// TwinCAT 3 PLC project ST710
// ProgramVersion: 3.1.4024.0
// libraries:
//   Tc2_Standard, * (Beckhoff Automation GmbH)
//   Tc2_System, * (Beckhoff Automation GmbH)
//   Tc3_Module, * (Beckhoff Automation GmbH)
// project tree:
//   DUTs/ Cyl_Module_DUT.TcDUT
//   / GlobalTextList.TcGTLO, PlcTask.TcTTO, Visualization Manager.TcVMO (not stored)
//   GVLs/ Alarm_DB.TcGVL, Auto_Seq_DB.TcGVL, Home_Seq_DB.TcGVL, Inputs.TcGVL, Outputs.TcGVL, Stn710_DB.TcGVL
//   POUs/ Auto_Sequence.TcPOU, HomeSequence.TcPOU, MAIN.TcPOU, Alarms.TcPOU, Robot.TcPOU, Module_call.TcPOU, PowerOn.TcPOU, RollerDoor.TcPOU, Trunion.TcPOU, TurnTable.TcPOU
//   POUs/Library/ Seq_list.TcTLO, FB_CylinderModule.TcPOU, Feedback_FB.TcPOU, Alarm_list.TcTLO
//   VISUs/ Visualization.TcVIS
// real-time tasks:
//   TASK PlcTask: cycle T#10ms, priority 20, ADS port 350

CONFIGURATION ST710
    RESOURCE PLC ON TwinCAT3
        TASK PlcTask(INTERVAL := T#10ms, PRIORITY := 20);
        PROGRAM MAIN WITH PlcTask : MAIN;
    END_RESOURCE
END_CONFIGURATION

// ---- DUTs/Cyl_Module_DUT.TcDUT
TYPE Cyl_Module_DUT :
STRUCT
	ResetFaults:BOOL;//Reset Fault CMD
    WorkCmd:BOOL ;//Cyl Work Postion CMD
    HomeCmd:BOOL ;//Cyl Home Postion CMD
    WorkSen:BOOL ;// Cyl Work Postion Input
    HomeSen:BOOL ;// Cyl Home Postion Input
    WorkCleartoMove:BOOL ;// Condition Healthy then 1
    HomeCleartoMove:BOOL ;// Condition Healthy then 1
    TimeoutValue:TIME ;// Time Required E.gT#500MS,T#2S
	ENO   : BOOL; //  Block Enable
	WorkSol    : BOOL; // Cyl Work Position Sol Output
    HomeSol: BOOL; //Cyl Home Position Sol Output
    WorkOver: BOOL; // Cyl AT Work Position
    HomeOver: BOOL; //Cyl AT Home Position
    ErrHomeInterlock: BOOL; //homeCleartoMove is low AND home command is active.
    ErrHomeTout: BOOL; //cylinder did NOT reachhome position within definedTIME
    ErrWorkInterlock: BOOL; //WorkCleartoMove is low AND work command is active.
    ErrWorkTout: BOOL; //cylinder did NOT reachwork position within definedtime
END_STRUCT
END_TYPE

// ---- GVLs/Alarm_DB.TcGVL
{attribute 'qualified_only'}
VAR_GLOBAL
	EMR_Stop_pressed : BOOL;
END_VAR

// ---- GVLs/Auto_Seq_DB.TcGVL
{attribute 'qualified_only'}
VAR_GLOBAL
	MHomeCycleStart		:BOOL;
	MWELD_RobotStart	:BOOL;
	M_MH_RobotStart		:BOOL;
	MCycleRun			:BOOL;
	MRollerDoor_CLOSE	:BOOL;
	MRollerDoor_Open	:BOOL;
	MTrunion_Move_0		:BOOL;
	MTrunion_Move_20	:BOOL;
	MTrunion_Move_45	:BOOL;
	MTrunion_Move_80	:BOOL;
	MClampClsGroup1		:BOOL;
	MClampClsGroup2		:BOOL;
	MTurntable_0		:BOOL;
	MTurntable_180		:BOOL;
	MClampOpenGrp1		:BOOL;
	MClampOpenGrp2		:BOOL;
	MStep				:INT;
	Part_Sensor1		:BOOL;
	Part_Sensor2		:BOOL;
	Part_Sensor3		:BOOL;
	Part_Sensor4		:BOOL;
END_VAR

// ---- GVLs/Home_Seq_DB.TcGVL
{attribute 'qualified_only'}
VAR_GLOBAL
	M_Group1ClampOpen :BOOL;
	M_Group2ClampOpen :BOOL;
	M_TT_0 : BOOL;
	M_Trunion_0 : BOOL;
	M_Door_Cls : BOOL;
	M_HomeDone : Bool;
END_VAR

// ---- GVLs/Inputs.TcGVL
{attribute 'qualified_only'}
VAR_GLOBAL
	Control_Pressure_Sw_In1_BPB1	: BOOL ;
	Control_Pressure_Sw_In2_BPB1	: BOOL ;
	Valve_Pos_BGB1					: BOOL ;
	CC6_Clamp_1_Sensor_HP			: BOOL ;
	CC6_Clamp_1_Sensor_WP			: BOOL ;
	CC4_Clamp_3_Sensor_HP			: BOOL ;
	CC4_Clamp_3_Sensor_WP			: BOOL ;
	CC4_Clamp_2_Sensor_HP			: BOOL ;
	CC4_Clamp_2_Sensor_WP			: BOOL ;
	CC4_Clamp_1_Sensor_HP			: BOOL ;
	CC4_Clamp_1_Sensor_WP			: BOOL ;
	CC2_Clamp_3_Sensor_HP			: BOOL ;
	CC2_Clamp_3_Sensor_WP			: BOOL ;
	CC3_Clamp_3_Sensor_HP			: BOOL ;
	CC3_Clamp_3_Sensor_WP			: BOOL ;
	CC3_Clamp_2_Sensor_HP			: BOOL ;
	CC3_Clamp_2_Sensor_WP			: BOOL ;
	CC3_Clamp_1_Sensor_HP			: BOOL ;
	CC3_Clamp_1_Sensor_WP			: BOOL ;
	CC1_Clamp_3_Sensor_HP			: BOOL ;
	CC1_Clamp_3_Sensor_WP			: BOOL ;
	CC1_Clamp_2_Sensor_HP			: BOOL ;
	CC1_Clamp_2_Sensor_WP			: BOOL ;
	CC1_Clamp_1_Sensor_HP			: BOOL ;
	CC1_Clamp_1_Sensor_WP			: BOOL ;
	CC2_Clamp_2_Sensor_HP			: BOOL ;
	CC2_Clamp_2_Sensor_WP			: BOOL ;
	CC2_Clamp_1_Sensor_HP			: BOOL ;
	CC2_Clamp_1_Sensor_WP			: BOOL ;
	CC5_Clamp_1_Sensor_HP			: BOOL ;
	CC5_Clamp_1_Sensor_WP			: BOOL ;
	PART_CONTROL_B13				: BOOL ;
	PART_CONTROL_B27				: BOOL ;
	PART_CONTROL_B14				: BOOL ;
	PART_CONTROL_B28				: BOOL ;
	PART_CONTROL_B12				: BOOL ;
	PART_CONTROL_B26				: BOOL ;
	PART_CONTROL_B11				: BOOL ;
	PART_CONTROL_B25				: BOOL ;
	PART_CONTROL_B10				: BOOL ;
	PART_CONTROL_B24				: BOOL ;
	PART_CONTROL_B7					: BOOL ;
	PART_CONTROL_B21				: BOOL ;
	PART_CONTROL_B6					: BOOL ;
	PART_CONTROL_B20				: BOOL ;
	PART_CONTROL_B5					: BOOL ;
	PART_CONTROL_B19				: BOOL ;
	PART_CONTROL_B4			 		: BOOL ;
	PART_CONTROL_B18				: BOOL ;
	PART_CONTROL_B3					: BOOL ;
	PART_CONTROL_B17				: BOOL ;
	PART_CONTROL_B2					: BOOL ;
	PART_CONTROL_B9					: BOOL ;
	PART_CONTROL_B23				: BOOL ;
	PART_CONTROL_B8					: BOOL ;
	PART_CONTROL_B22				: BOOL ;
	iEMR_Stop_PB					: BOOL ;
	iControl_On						: BOOL ;
	iControl_Off					: BOOL ;
	iAuto_Manual					: BOOL ;
	iResetFault 					: BOOL ;
	iCycle_start					:BOOL;
	iPalm_Button					:BOOL;
	
END_VAR

// ---- GVLs/Outputs.TcGVL
{attribute 'qualified_only'}
VAR_GLOBAL
	CC1_CLAMPING_UNIT1_3_WP			: BOOL ;
	CC1_CLAMPING_UNIT1_3_HP			: BOOL ;
	CC2_CLAMPING_UNIT2_3_WP			: BOOL ;
	CC2_CLAMPING_UNIT2_3_HP			: BOOL ;
	CC3_CLAMPING_UNIT3_3_WP			: BOOL ;
	CC3_CLAMPING_UNIT3_3_HP			: BOOL ;
	CC4_CLAMPING_UNIT4_3_WP			: BOOL ;
	CC4_CLAMPING_UNIT4_3_HP			: BOOL ;
	CC5_CLAMPING_UNIT5_1_WP			: BOOL ;
	CC5_CLAMPING_UNIT5_1_HP			: BOOL ;
	CC6_CLAMPING_UNIT6_1_WP			: BOOL ;
	CC6_CLAMPING_UNIT6_1_HP			: BOOL ;
	qPower_On						: BOOL ;
	qStnAuto						: BOOL ;
	qStnMan							: BOOL ;
END_VAR

// ---- GVLs/Stn710_DB.TcGVL
{attribute 'qualified_only'}
VAR_GLOBAL
	M_TT_MotorRun  : BOOL;
	M_TT_MotorDir  : BOOL;
	M_TT_CW		   : BOOL;
	M_TT_CCW		: BOOL;
	M_TT_FwdSens	: BOOL;
	M_TT_RevSens	: BOOL;
	M_TR_Motor0  	: BOOL;
	M_TR_Motor20  	: BOOL;
	M_TR_Motor45  	: BOOL;
	M_TR_Motor80  	: BOOL;
	M_TR_0_FB		: BOOL;
	M_TR_20_FB		: BOOL;
	M_TR_45_FB		: BOOL;
	M_TR_80_FB		: BOOL;
	M_TR_0_CMD		: BOOL;
	M_TR_20_CMD		: BOOL;
	M_TR_45_CMD		: BOOL;
	M_TR_80_CMD		: BOOL;
	MQ_DR_UP	  	: BOOL;
	MQ_DR_DOWN  	: BOOL;
	M_DR_UP		   	: BOOL;
	M_DR_DOWN		: BOOL;
	M_DR_UPSens		: BOOL;
	M_DR_DNSens		: BOOL;
	MH_RobotHome	: BOOL;
	MH_RobotBusy	: BOOL;
	MH_RobotDone	: BOOL;
	WELD_RobotHome	: BOOL;
	WELD_RobotBusy	: BOOL;
	WELD_RobotDone	: BOOL;
	Alarm_count : INT;
	CC1_CLAMP : Cyl_Module_DUT;
	CC2_CLAMP : Cyl_Module_DUT;
	CC3_CLAMP : Cyl_Module_DUT;
	CC4_CLAMP : Cyl_Module_DUT;
	CC5_CLAMP : Cyl_Module_DUT;
	CC6_CLAMP : Cyl_Module_DUT;	
END_VAR

// ---- POUs/MAIN.TcPOU
PROGRAM MAIN
VAR
	Modules: Module_call;
	tAlwaysOn: BOOL; //Temporary BIT FOR Always On
    tAlwaysOff: BOOL; //Temporary BIT FOR Always Off
END_VAR

VAR CONSTANT
END_VAR

// Always ON Logic
tAlwaysOn := TRUE;

// Module call
Modules();

END_PROGRAM

// ---- POUs/Module_call.TcPOU
FUNCTION_BLOCK Module_call
VAR_INPUT
END_VAR
VAR_OUTPUT
END_VAR
VAR
	CC1_UNIT1_3_Cyl: FB_CylinderModule;	
	CC2_UNIT2_3_Cyl: FB_CylinderModule;
	CC3_UNIT3_3_Cyl: FB_CylinderModule;
	CC4_UNIT4_3_Cyl: FB_CylinderModule;
	CC5_UNIT5_1_Cyl: FB_CylinderModule;
	CC6_UNIT6_1_Cyl: FB_CylinderModule;
	CC1_Feedback_FB: Feedback_FB;
	CC2_Feedback_FB: Feedback_FB;
	CC3_Feedback_FB: Feedback_FB;
	CC4_Feedback_FB: Feedback_FB;
	CC5_Feedback_FB: Feedback_FB;
	CC6_Feedback_FB: Feedback_FB;
	CC1_Feedback_1: BOOL;
	CC1_Feedback_2: BOOL;
	CC2_Feedback_1: BOOL;
	CC2_Feedback_2: BOOL;
	CC3_Feedback_1: BOOL;
	CC3_Feedback_2: BOOL;
	CC4_Feedback_1: BOOL;
	CC4_Feedback_2: BOOL;
	PowerOn: PowerOn;
	TurnTable_0: TurnTable;
	TT_Feedback_FB: Feedback_FB;
	Trunion_0: Trunion;
	Tr_Feedback_FB: Feedback_FB;
	RollerDoor_0: RollerDoor;
	Door_Feedback_FB: Feedback_FB;
	MH_Robot: Robot;
	Weld_Robot: Robot;
	Auto_Sequence_0: Auto_Sequence;
	TR_Feedback_FB1: Feedback_FB;
	HomeSequence_0: HomeSequence;
	Alarms_0: Alarms;
END_VAR
VAR // added by the converter: edge detectors and wires of the graphical bodies
    _w1, _w2, _w3, _w4, _w5, _w6, _w7, _w8 : BOOL;
END_VAR

// note: this text did not pass the execution check against the stored diagram
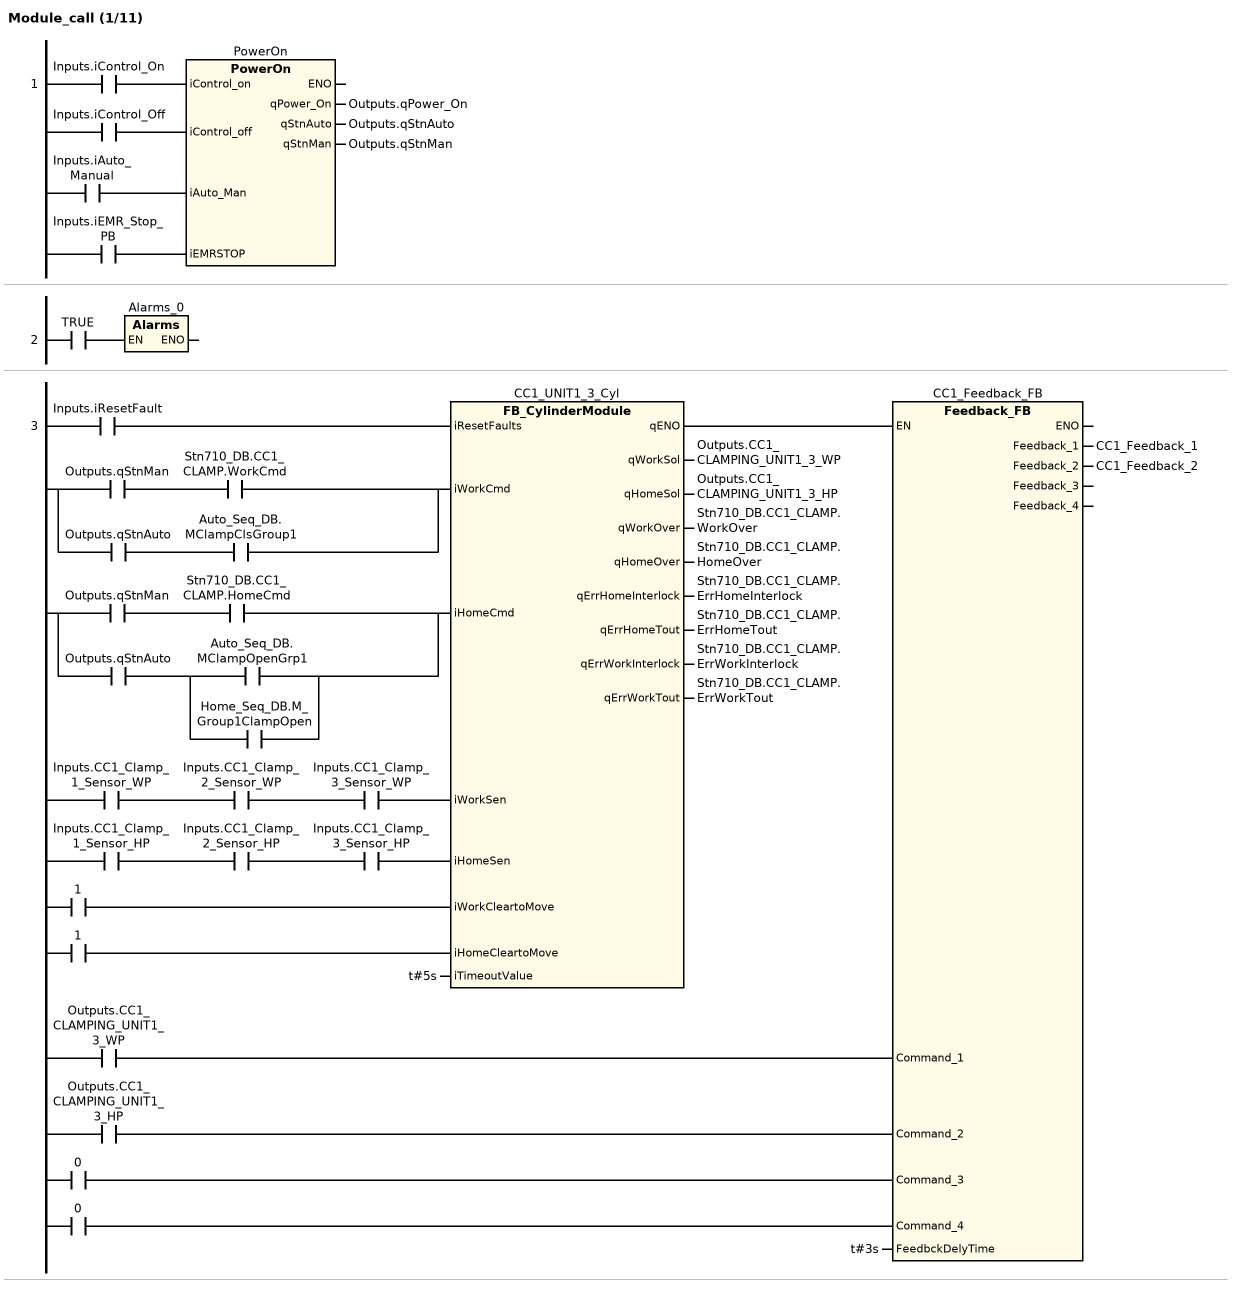
// NETWORK 1
PowerOn(
    iControl_on := Inputs.iControl_On,
    iControl_off := Inputs.iControl_Off,
    iAuto_Man := Inputs.iAuto_Manual,
    iEMRSTOP := Inputs.iEMR_Stop_PB,
    qPower_On => Outputs.qPower_On,
    qStnAuto => Outputs.qStnAuto,
    qStnMan => Outputs.qStnMan);

// NETWORK 2
Alarms_0(EN := TRUE); // Alarms

// NETWORK 3
CC1_UNIT1_3_Cyl(
    iResetFaults := Inputs.iResetFault,
    iWorkCmd := Outputs.qStnMan AND Stn710_DB.CC1_CLAMP.WorkCmd OR Outputs.qStnAuto AND Auto_Seq_DB.MClampClsGroup1,
    iHomeCmd := Outputs.qStnMan AND Stn710_DB.CC1_CLAMP.HomeCmd OR Outputs.qStnAuto AND (Auto_Seq_DB.MClampOpenGrp1 OR Home_Seq_DB.M_Group1ClampOpen),
    iWorkSen := Inputs.CC1_Clamp_1_Sensor_WP AND Inputs.CC1_Clamp_2_Sensor_WP AND Inputs.CC1_Clamp_3_Sensor_WP,
    iHomeSen := Inputs.CC1_Clamp_1_Sensor_HP AND Inputs.CC1_Clamp_2_Sensor_HP AND Inputs.CC1_Clamp_3_Sensor_HP,
    iWorkCleartoMove := 1,
    iHomeCleartoMove := 1,
    iTimeoutValue := t#5s,
    qWorkSol => Outputs.CC1_CLAMPING_UNIT1_3_WP,
    qHomeSol => Outputs.CC1_CLAMPING_UNIT1_3_HP,
    qWorkOver => Stn710_DB.CC1_CLAMP.WorkOver,
    qHomeOver => Stn710_DB.CC1_CLAMP.HomeOver,
    qErrHomeInterlock => Stn710_DB.CC1_CLAMP.ErrHomeInterlock,
    qErrHomeTout => Stn710_DB.CC1_CLAMP.ErrHomeTout,
    qErrWorkInterlock => Stn710_DB.CC1_CLAMP.ErrWorkInterlock,
    qErrWorkTout => Stn710_DB.CC1_CLAMP.ErrWorkTout); // FB_CylinderModule
CC1_Feedback_FB(
    EN := CC1_UNIT1_3_Cyl.qENO,
    Command_1 := Outputs.CC1_CLAMPING_UNIT1_3_WP,
    Command_2 := Outputs.CC1_CLAMPING_UNIT1_3_HP,
    Command_3 := 0,
    Command_4 := 0,
    FeedbckDelyTime := t#3s,
    Feedback_1 => CC1_Feedback_1,
    Feedback_2 => CC1_Feedback_2); // Feedback_FB

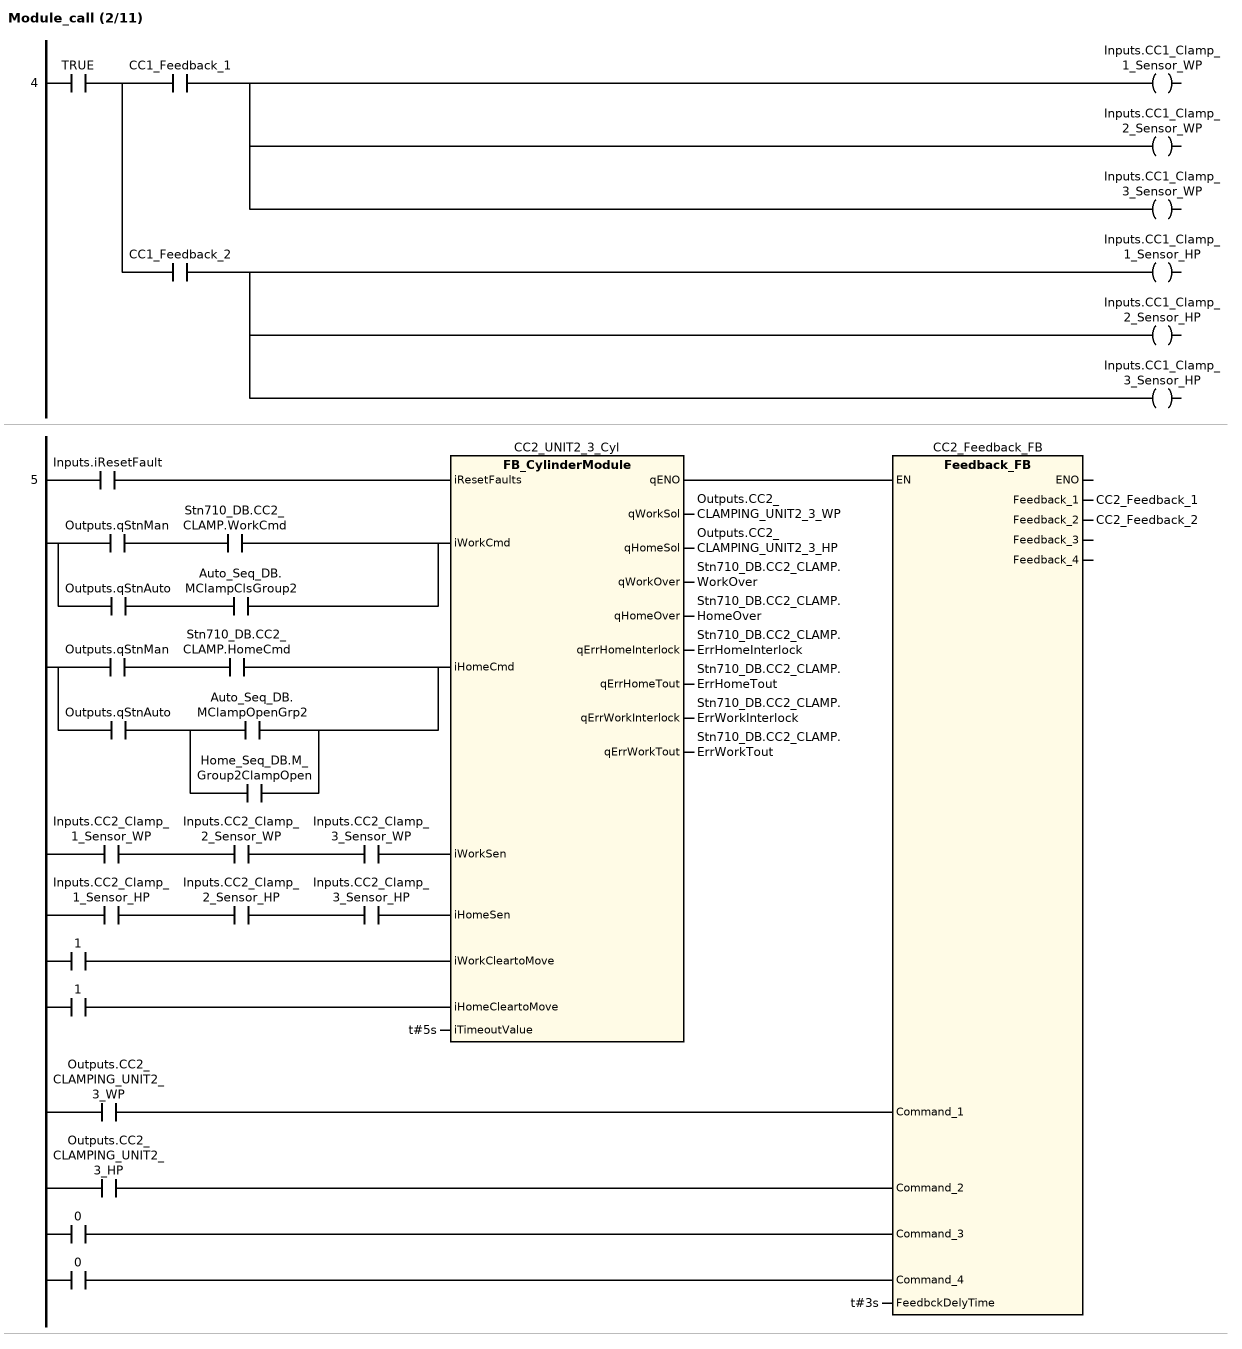
// NETWORK 4
_w1 := TRUE AND CC1_Feedback_1;
Inputs.CC1_Clamp_1_Sensor_WP := _w1;
Inputs.CC1_Clamp_2_Sensor_WP := _w1;
Inputs.CC1_Clamp_3_Sensor_WP := _w1;
_w2 := TRUE AND CC1_Feedback_2;
Inputs.CC1_Clamp_1_Sensor_HP := _w2;
Inputs.CC1_Clamp_2_Sensor_HP := _w2;
Inputs.CC1_Clamp_3_Sensor_HP := _w2;

// NETWORK 5
CC2_UNIT2_3_Cyl(
    iResetFaults := Inputs.iResetFault,
    iWorkCmd := Outputs.qStnMan AND Stn710_DB.CC2_CLAMP.WorkCmd OR Outputs.qStnAuto AND Auto_Seq_DB.MClampClsGroup2,
    iHomeCmd := Outputs.qStnMan AND Stn710_DB.CC2_CLAMP.HomeCmd OR Outputs.qStnAuto AND (Auto_Seq_DB.MClampOpenGrp2 OR Home_Seq_DB.M_Group2ClampOpen),
    iWorkSen := Inputs.CC2_Clamp_1_Sensor_WP AND Inputs.CC2_Clamp_2_Sensor_WP AND Inputs.CC2_Clamp_3_Sensor_WP,
    iHomeSen := Inputs.CC2_Clamp_1_Sensor_HP AND Inputs.CC2_Clamp_2_Sensor_HP AND Inputs.CC2_Clamp_3_Sensor_HP,
    iWorkCleartoMove := 1,
    iHomeCleartoMove := 1,
    iTimeoutValue := t#5s,
    qWorkSol => Outputs.CC2_CLAMPING_UNIT2_3_WP,
    qHomeSol => Outputs.CC2_CLAMPING_UNIT2_3_HP,
    qWorkOver => Stn710_DB.CC2_CLAMP.WorkOver,
    qHomeOver => Stn710_DB.CC2_CLAMP.HomeOver,
    qErrHomeInterlock => Stn710_DB.CC2_CLAMP.ErrHomeInterlock,
    qErrHomeTout => Stn710_DB.CC2_CLAMP.ErrHomeTout,
    qErrWorkInterlock => Stn710_DB.CC2_CLAMP.ErrWorkInterlock,
    qErrWorkTout => Stn710_DB.CC2_CLAMP.ErrWorkTout); // FB_CylinderModule
CC2_Feedback_FB(
    EN := CC2_UNIT2_3_Cyl.qENO,
    Command_1 := Outputs.CC2_CLAMPING_UNIT2_3_WP,
    Command_2 := Outputs.CC2_CLAMPING_UNIT2_3_HP,
    Command_3 := 0,
    Command_4 := 0,
    FeedbckDelyTime := t#3s,
    Feedback_1 => CC2_Feedback_1,
    Feedback_2 => CC2_Feedback_2); // Feedback_FB

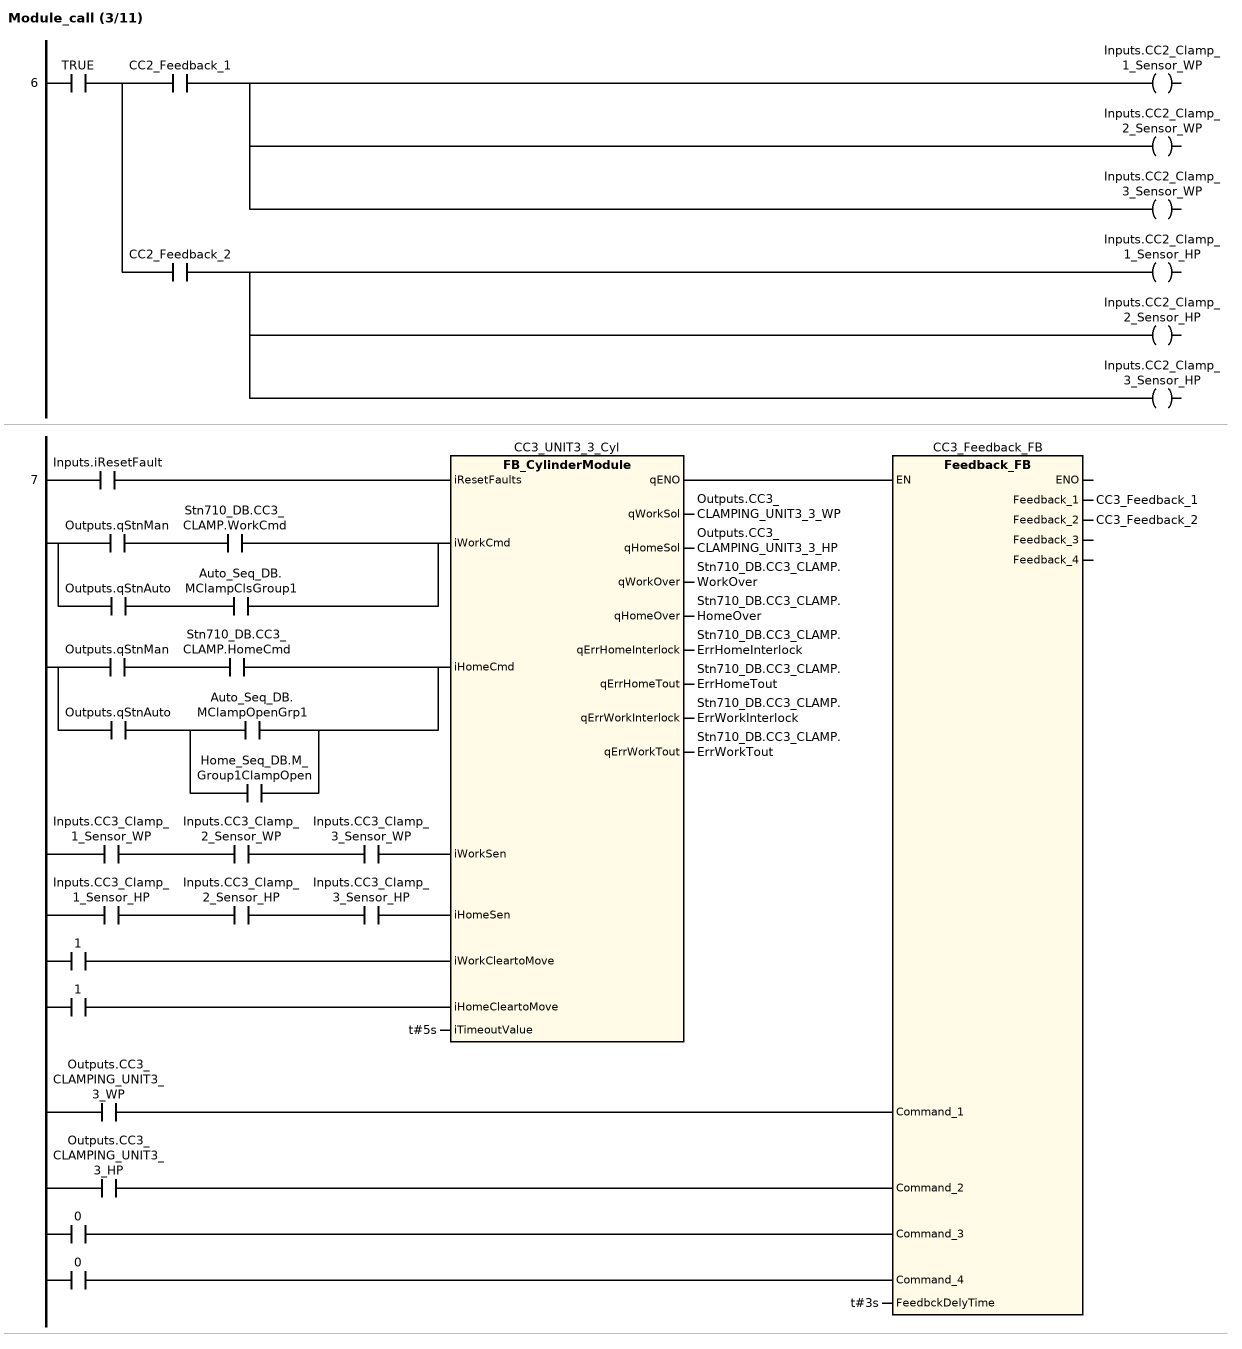
// NETWORK 6
_w3 := TRUE AND CC2_Feedback_1;
Inputs.CC2_Clamp_1_Sensor_WP := _w3;
Inputs.CC2_Clamp_2_Sensor_WP := _w3;
Inputs.CC2_Clamp_3_Sensor_WP := _w3;
_w4 := TRUE AND CC2_Feedback_2;
Inputs.CC2_Clamp_1_Sensor_HP := _w4;
Inputs.CC2_Clamp_2_Sensor_HP := _w4;
Inputs.CC2_Clamp_3_Sensor_HP := _w4;

// NETWORK 7
CC3_UNIT3_3_Cyl(
    iResetFaults := Inputs.iResetFault,
    iWorkCmd := Outputs.qStnMan AND Stn710_DB.CC3_CLAMP.WorkCmd OR Outputs.qStnAuto AND Auto_Seq_DB.MClampClsGroup1,
    iHomeCmd := Outputs.qStnMan AND Stn710_DB.CC3_CLAMP.HomeCmd OR Outputs.qStnAuto AND (Auto_Seq_DB.MClampOpenGrp1 OR Home_Seq_DB.M_Group1ClampOpen),
    iWorkSen := Inputs.CC3_Clamp_1_Sensor_WP AND Inputs.CC3_Clamp_2_Sensor_WP AND Inputs.CC3_Clamp_3_Sensor_WP,
    iHomeSen := Inputs.CC3_Clamp_1_Sensor_HP AND Inputs.CC3_Clamp_2_Sensor_HP AND Inputs.CC3_Clamp_3_Sensor_HP,
    iWorkCleartoMove := 1,
    iHomeCleartoMove := 1,
    iTimeoutValue := t#5s,
    qWorkSol => Outputs.CC3_CLAMPING_UNIT3_3_WP,
    qHomeSol => Outputs.CC3_CLAMPING_UNIT3_3_HP,
    qWorkOver => Stn710_DB.CC3_CLAMP.WorkOver,
    qHomeOver => Stn710_DB.CC3_CLAMP.HomeOver,
    qErrHomeInterlock => Stn710_DB.CC3_CLAMP.ErrHomeInterlock,
    qErrHomeTout => Stn710_DB.CC3_CLAMP.ErrHomeTout,
    qErrWorkInterlock => Stn710_DB.CC3_CLAMP.ErrWorkInterlock,
    qErrWorkTout => Stn710_DB.CC3_CLAMP.ErrWorkTout); // FB_CylinderModule
CC3_Feedback_FB(
    EN := CC3_UNIT3_3_Cyl.qENO,
    Command_1 := Outputs.CC3_CLAMPING_UNIT3_3_WP,
    Command_2 := Outputs.CC3_CLAMPING_UNIT3_3_HP,
    Command_3 := 0,
    Command_4 := 0,
    FeedbckDelyTime := t#3s,
    Feedback_1 => CC3_Feedback_1,
    Feedback_2 => CC3_Feedback_2); // Feedback_FB

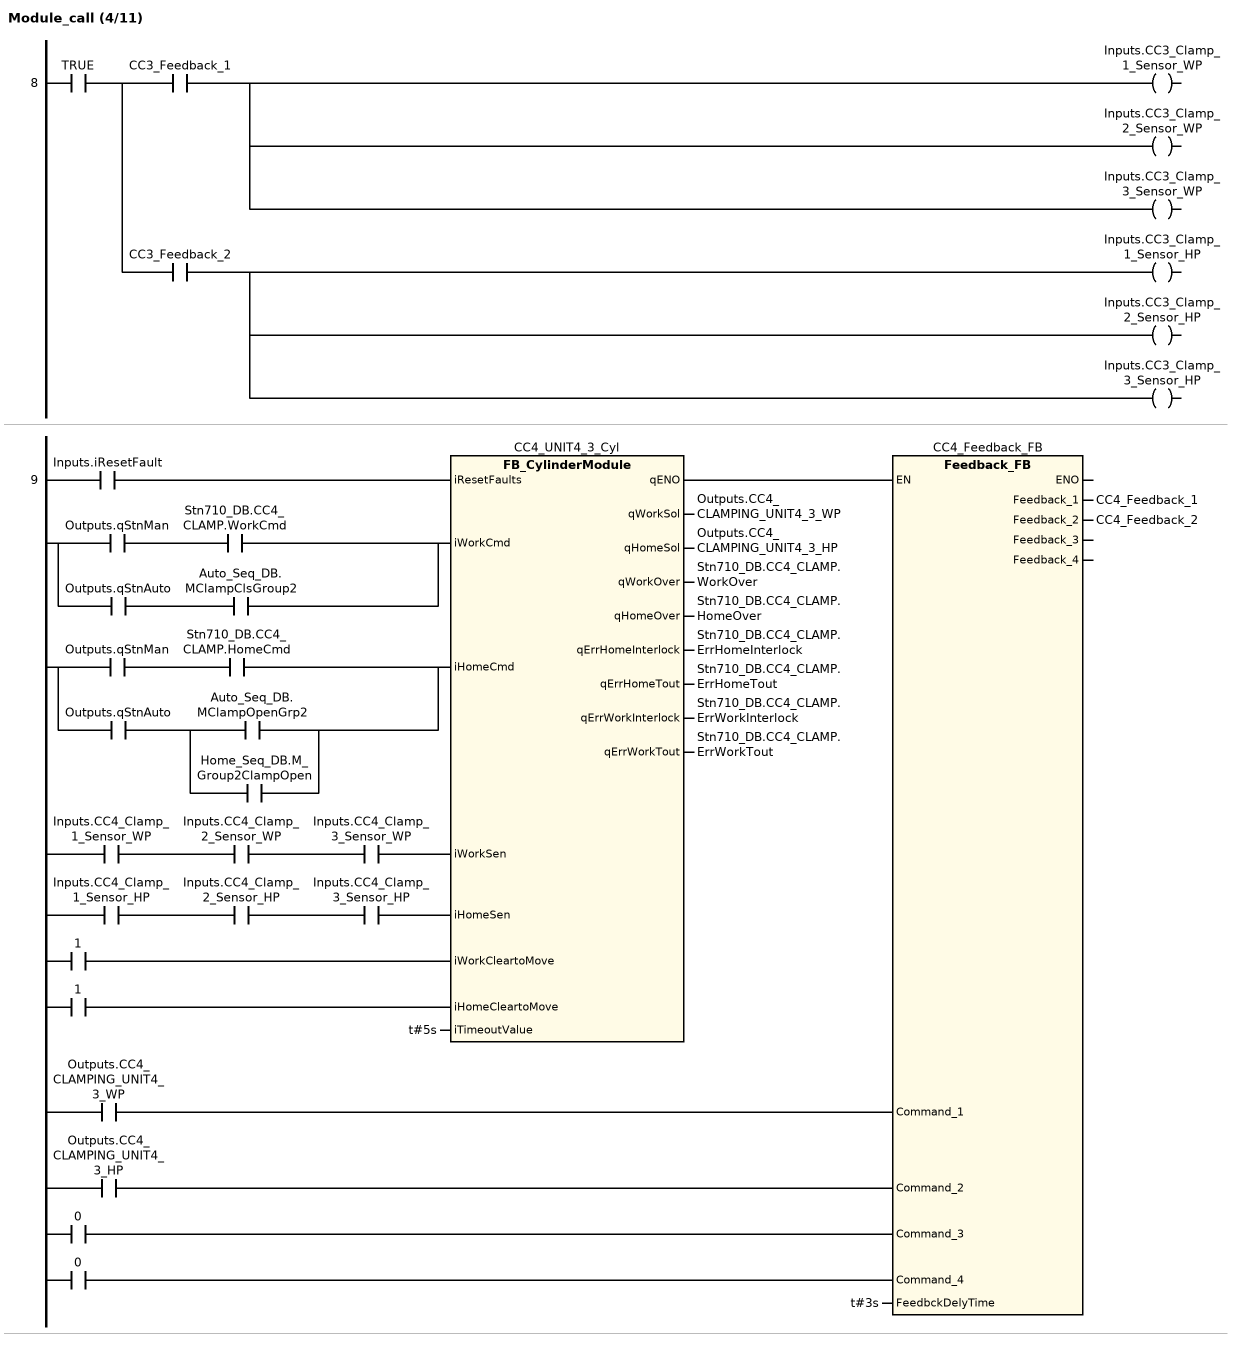
// NETWORK 8
_w5 := TRUE AND CC3_Feedback_1;
Inputs.CC3_Clamp_1_Sensor_WP := _w5;
Inputs.CC3_Clamp_2_Sensor_WP := _w5;
Inputs.CC3_Clamp_3_Sensor_WP := _w5;
_w6 := TRUE AND CC3_Feedback_2;
Inputs.CC3_Clamp_1_Sensor_HP := _w6;
Inputs.CC3_Clamp_2_Sensor_HP := _w6;
Inputs.CC3_Clamp_3_Sensor_HP := _w6;

// NETWORK 9
CC4_UNIT4_3_Cyl(
    iResetFaults := Inputs.iResetFault,
    iWorkCmd := Outputs.qStnMan AND Stn710_DB.CC4_CLAMP.WorkCmd OR Outputs.qStnAuto AND Auto_Seq_DB.MClampClsGroup2,
    iHomeCmd := Outputs.qStnMan AND Stn710_DB.CC4_CLAMP.HomeCmd OR Outputs.qStnAuto AND (Auto_Seq_DB.MClampOpenGrp2 OR Home_Seq_DB.M_Group2ClampOpen),
    iWorkSen := Inputs.CC4_Clamp_1_Sensor_WP AND Inputs.CC4_Clamp_2_Sensor_WP AND Inputs.CC4_Clamp_3_Sensor_WP,
    iHomeSen := Inputs.CC4_Clamp_1_Sensor_HP AND Inputs.CC4_Clamp_2_Sensor_HP AND Inputs.CC4_Clamp_3_Sensor_HP,
    iWorkCleartoMove := 1,
    iHomeCleartoMove := 1,
    iTimeoutValue := t#5s,
    qWorkSol => Outputs.CC4_CLAMPING_UNIT4_3_WP,
    qHomeSol => Outputs.CC4_CLAMPING_UNIT4_3_HP,
    qWorkOver => Stn710_DB.CC4_CLAMP.WorkOver,
    qHomeOver => Stn710_DB.CC4_CLAMP.HomeOver,
    qErrHomeInterlock => Stn710_DB.CC4_CLAMP.ErrHomeInterlock,
    qErrHomeTout => Stn710_DB.CC4_CLAMP.ErrHomeTout,
    qErrWorkInterlock => Stn710_DB.CC4_CLAMP.ErrWorkInterlock,
    qErrWorkTout => Stn710_DB.CC4_CLAMP.ErrWorkTout); // FB_CylinderModule
CC4_Feedback_FB(
    EN := CC4_UNIT4_3_Cyl.qENO,
    Command_1 := Outputs.CC4_CLAMPING_UNIT4_3_WP,
    Command_2 := Outputs.CC4_CLAMPING_UNIT4_3_HP,
    Command_3 := 0,
    Command_4 := 0,
    FeedbckDelyTime := t#3s,
    Feedback_1 => CC4_Feedback_1,
    Feedback_2 => CC4_Feedback_2); // Feedback_FB

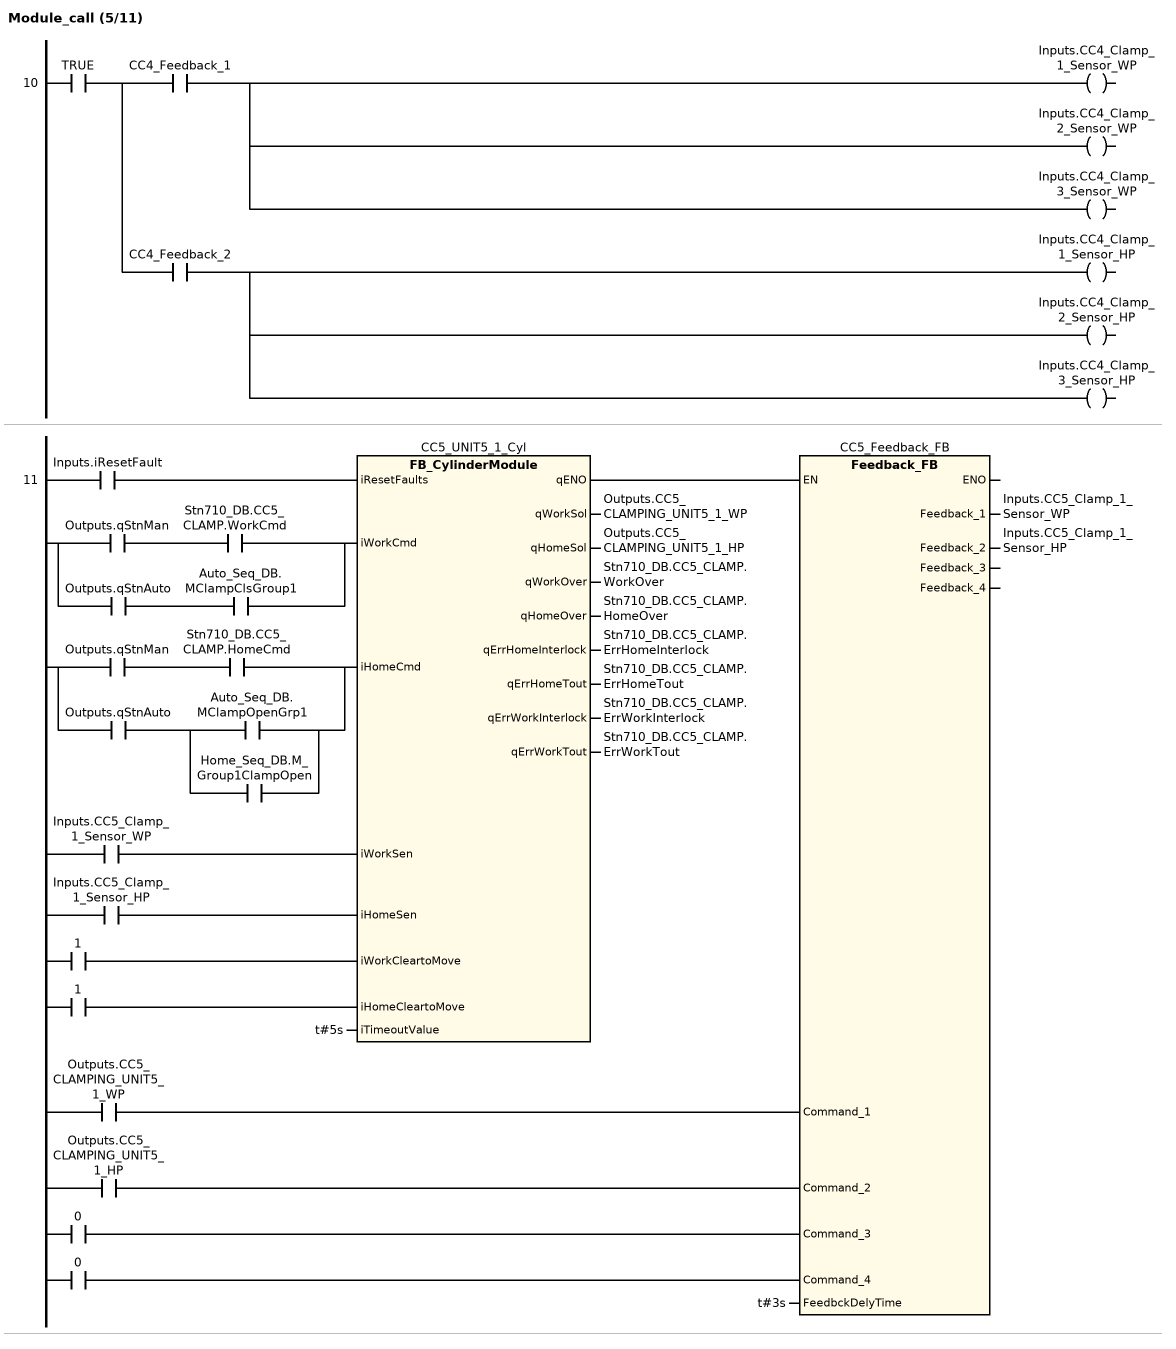
// NETWORK 10
_w7 := TRUE AND CC4_Feedback_1;
Inputs.CC4_Clamp_1_Sensor_WP := _w7;
Inputs.CC4_Clamp_2_Sensor_WP := _w7;
Inputs.CC4_Clamp_3_Sensor_WP := _w7;
_w8 := TRUE AND CC4_Feedback_2;
Inputs.CC4_Clamp_1_Sensor_HP := _w8;
Inputs.CC4_Clamp_2_Sensor_HP := _w8;
Inputs.CC4_Clamp_3_Sensor_HP := _w8;

// NETWORK 11
CC5_UNIT5_1_Cyl(
    iResetFaults := Inputs.iResetFault,
    iWorkCmd := Outputs.qStnMan AND Stn710_DB.CC5_CLAMP.WorkCmd OR Outputs.qStnAuto AND Auto_Seq_DB.MClampClsGroup1,
    iHomeCmd := Outputs.qStnMan AND Stn710_DB.CC5_CLAMP.HomeCmd OR Outputs.qStnAuto AND (Auto_Seq_DB.MClampOpenGrp1 OR Home_Seq_DB.M_Group1ClampOpen),
    iWorkSen := Inputs.CC5_Clamp_1_Sensor_WP,
    iHomeSen := Inputs.CC5_Clamp_1_Sensor_HP,
    iWorkCleartoMove := 1,
    iHomeCleartoMove := 1,
    iTimeoutValue := t#5s,
    qWorkSol => Outputs.CC5_CLAMPING_UNIT5_1_WP,
    qHomeSol => Outputs.CC5_CLAMPING_UNIT5_1_HP,
    qWorkOver => Stn710_DB.CC5_CLAMP.WorkOver,
    qHomeOver => Stn710_DB.CC5_CLAMP.HomeOver,
    qErrHomeInterlock => Stn710_DB.CC5_CLAMP.ErrHomeInterlock,
    qErrHomeTout => Stn710_DB.CC5_CLAMP.ErrHomeTout,
    qErrWorkInterlock => Stn710_DB.CC5_CLAMP.ErrWorkInterlock,
    qErrWorkTout => Stn710_DB.CC5_CLAMP.ErrWorkTout); // FB_CylinderModule
CC5_Feedback_FB(
    EN := CC5_UNIT5_1_Cyl.qENO,
    Command_1 := Outputs.CC5_CLAMPING_UNIT5_1_WP,
    Command_2 := Outputs.CC5_CLAMPING_UNIT5_1_HP,
    Command_3 := 0,
    Command_4 := 0,
    FeedbckDelyTime := t#3s,
    Feedback_1 => Inputs.CC5_Clamp_1_Sensor_WP,
    Feedback_2 => Inputs.CC5_Clamp_1_Sensor_HP); // Feedback_FB

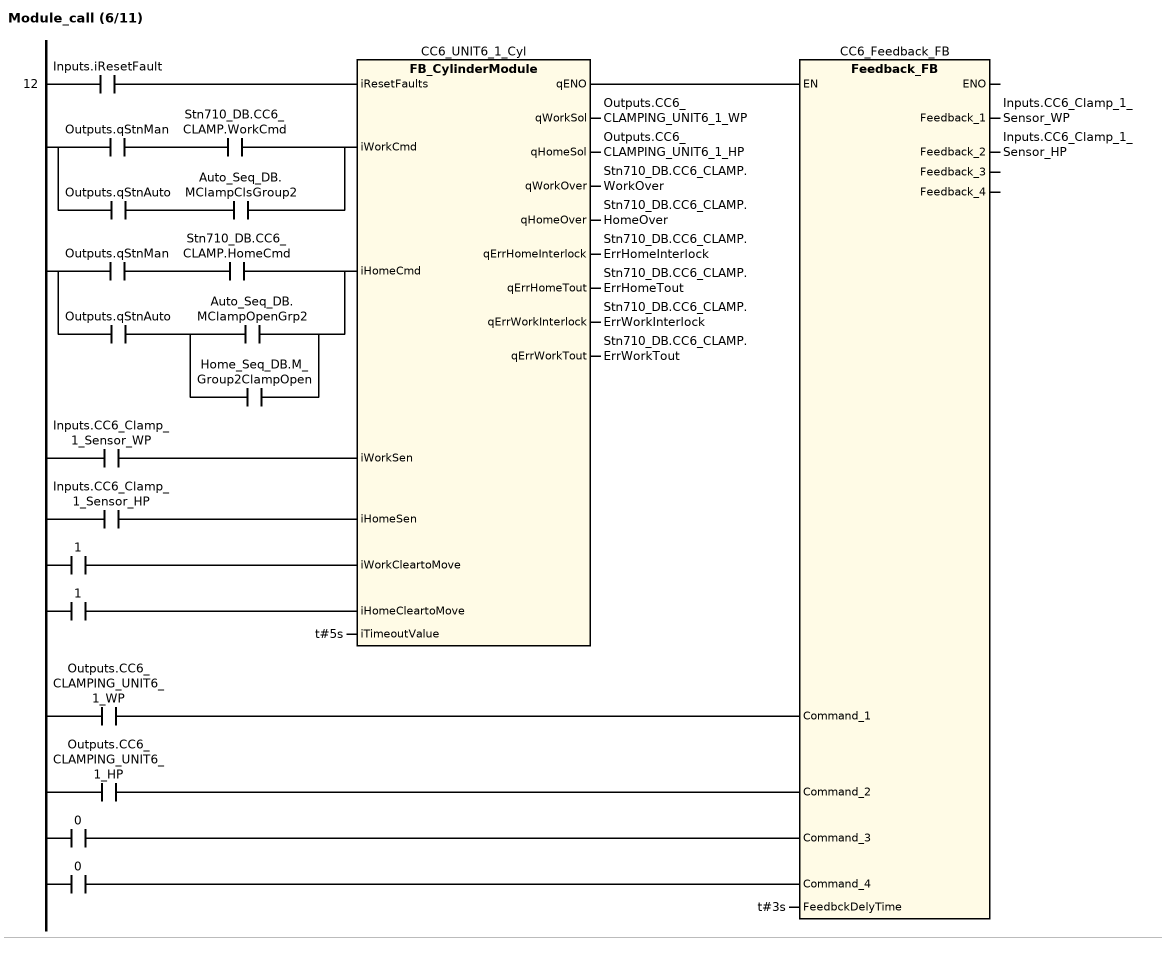
// NETWORK 12
CC6_UNIT6_1_Cyl(
    iResetFaults := Inputs.iResetFault,
    iWorkCmd := Outputs.qStnMan AND Stn710_DB.CC6_CLAMP.WorkCmd OR Outputs.qStnAuto AND Auto_Seq_DB.MClampClsGroup2,
    iHomeCmd := Outputs.qStnMan AND Stn710_DB.CC6_CLAMP.HomeCmd OR Outputs.qStnAuto AND (Auto_Seq_DB.MClampOpenGrp2 OR Home_Seq_DB.M_Group2ClampOpen),
    iWorkSen := Inputs.CC6_Clamp_1_Sensor_WP,
    iHomeSen := Inputs.CC6_Clamp_1_Sensor_HP,
    iWorkCleartoMove := 1,
    iHomeCleartoMove := 1,
    iTimeoutValue := t#5s,
    qWorkSol => Outputs.CC6_CLAMPING_UNIT6_1_WP,
    qHomeSol => Outputs.CC6_CLAMPING_UNIT6_1_HP,
    qWorkOver => Stn710_DB.CC6_CLAMP.WorkOver,
    qHomeOver => Stn710_DB.CC6_CLAMP.HomeOver,
    qErrHomeInterlock => Stn710_DB.CC6_CLAMP.ErrHomeInterlock,
    qErrHomeTout => Stn710_DB.CC6_CLAMP.ErrHomeTout,
    qErrWorkInterlock => Stn710_DB.CC6_CLAMP.ErrWorkInterlock,
    qErrWorkTout => Stn710_DB.CC6_CLAMP.ErrWorkTout); // FB_CylinderModule
CC6_Feedback_FB(
    EN := CC6_UNIT6_1_Cyl.qENO,
    Command_1 := Outputs.CC6_CLAMPING_UNIT6_1_WP,
    Command_2 := Outputs.CC6_CLAMPING_UNIT6_1_HP,
    Command_3 := 0,
    Command_4 := 0,
    FeedbckDelyTime := t#3s,
    Feedback_1 => Inputs.CC6_Clamp_1_Sensor_WP,
    Feedback_2 => Inputs.CC6_Clamp_1_Sensor_HP); // Feedback_FB

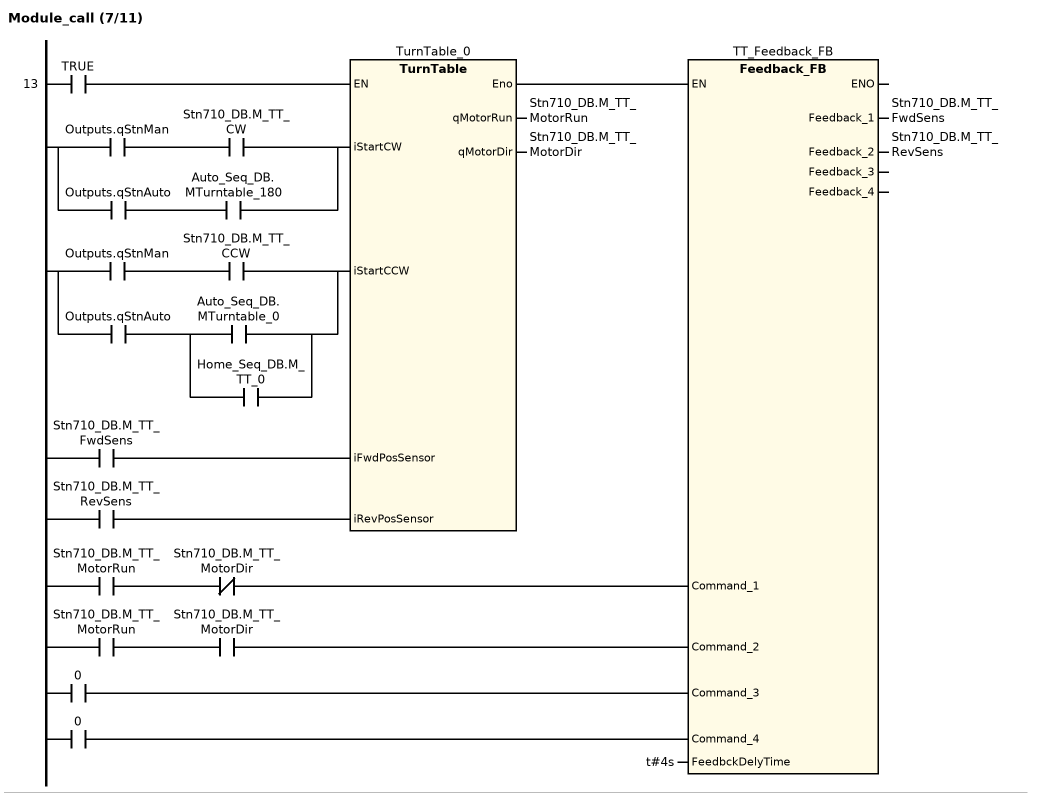
// NETWORK 13
TurnTable_0(
    EN := TRUE,
    iStartCW := Outputs.qStnMan AND Stn710_DB.M_TT_CW OR Outputs.qStnAuto AND Auto_Seq_DB.MTurntable_180,
    iStartCCW := Outputs.qStnMan AND Stn710_DB.M_TT_CCW OR Outputs.qStnAuto AND (Auto_Seq_DB.MTurntable_0 OR Home_Seq_DB.M_TT_0),
    iFwdPosSensor := Stn710_DB.M_TT_FwdSens,
    iRevPosSensor := Stn710_DB.M_TT_RevSens,
    qMotorRun => Stn710_DB.M_TT_MotorRun,
    qMotorDir => Stn710_DB.M_TT_MotorDir); // TurnTable
TT_Feedback_FB(
    EN := TRUE,
    Command_1 := Stn710_DB.M_TT_MotorRun AND NOT Stn710_DB.M_TT_MotorDir,
    Command_2 := Stn710_DB.M_TT_MotorRun AND Stn710_DB.M_TT_MotorDir,
    Command_3 := 0,
    Command_4 := 0,
    FeedbckDelyTime := t#4s,
    Feedback_1 => Stn710_DB.M_TT_FwdSens,
    Feedback_2 => Stn710_DB.M_TT_RevSens); // Feedback_FB

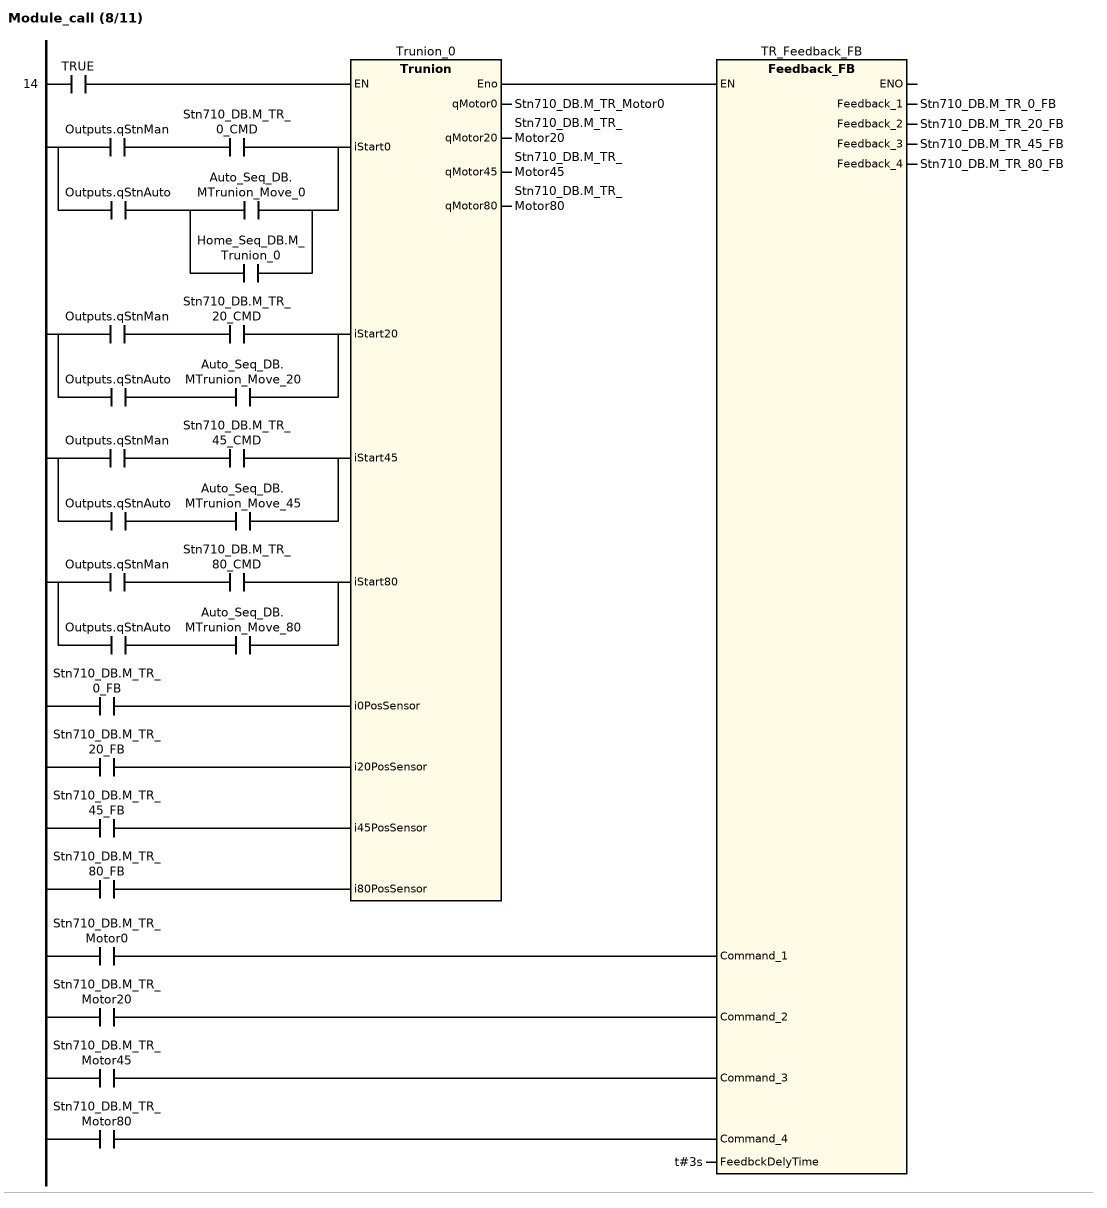
// NETWORK 14
Trunion_0(
    EN := TRUE,
    iStart0 := Outputs.qStnMan AND Stn710_DB.M_TR_0_CMD OR Outputs.qStnAuto AND (Auto_Seq_DB.MTrunion_Move_0 OR Home_Seq_DB.M_Trunion_0),
    iStart20 := Outputs.qStnMan AND Stn710_DB.M_TR_20_CMD OR Outputs.qStnAuto AND Auto_Seq_DB.MTrunion_Move_20,
    iStart45 := Outputs.qStnMan AND Stn710_DB.M_TR_45_CMD OR Outputs.qStnAuto AND Auto_Seq_DB.MTrunion_Move_45,
    iStart80 := Outputs.qStnMan AND Stn710_DB.M_TR_80_CMD OR Outputs.qStnAuto AND Auto_Seq_DB.MTrunion_Move_80,
    i0PosSensor := Stn710_DB.M_TR_0_FB,
    i20PosSensor := Stn710_DB.M_TR_20_FB,
    i45PosSensor := Stn710_DB.M_TR_45_FB,
    i80PosSensor := Stn710_DB.M_TR_80_FB,
    qMotor0 => Stn710_DB.M_TR_Motor0,
    qMotor20 => Stn710_DB.M_TR_Motor20,
    qMotor45 => Stn710_DB.M_TR_Motor45,
    qMotor80 => Stn710_DB.M_TR_Motor80); // Trunion
TR_Feedback_FB(
    EN := TRUE,
    Command_1 := Stn710_DB.M_TR_Motor0,
    Command_2 := Stn710_DB.M_TR_Motor20,
    Command_3 := Stn710_DB.M_TR_Motor45,
    Command_4 := Stn710_DB.M_TR_Motor80,
    FeedbckDelyTime := t#3s,
    Feedback_1 => Stn710_DB.M_TR_0_FB,
    Feedback_2 => Stn710_DB.M_TR_20_FB,
    Feedback_3 => Stn710_DB.M_TR_45_FB,
    Feedback_4 => Stn710_DB.M_TR_80_FB); // Feedback_FB

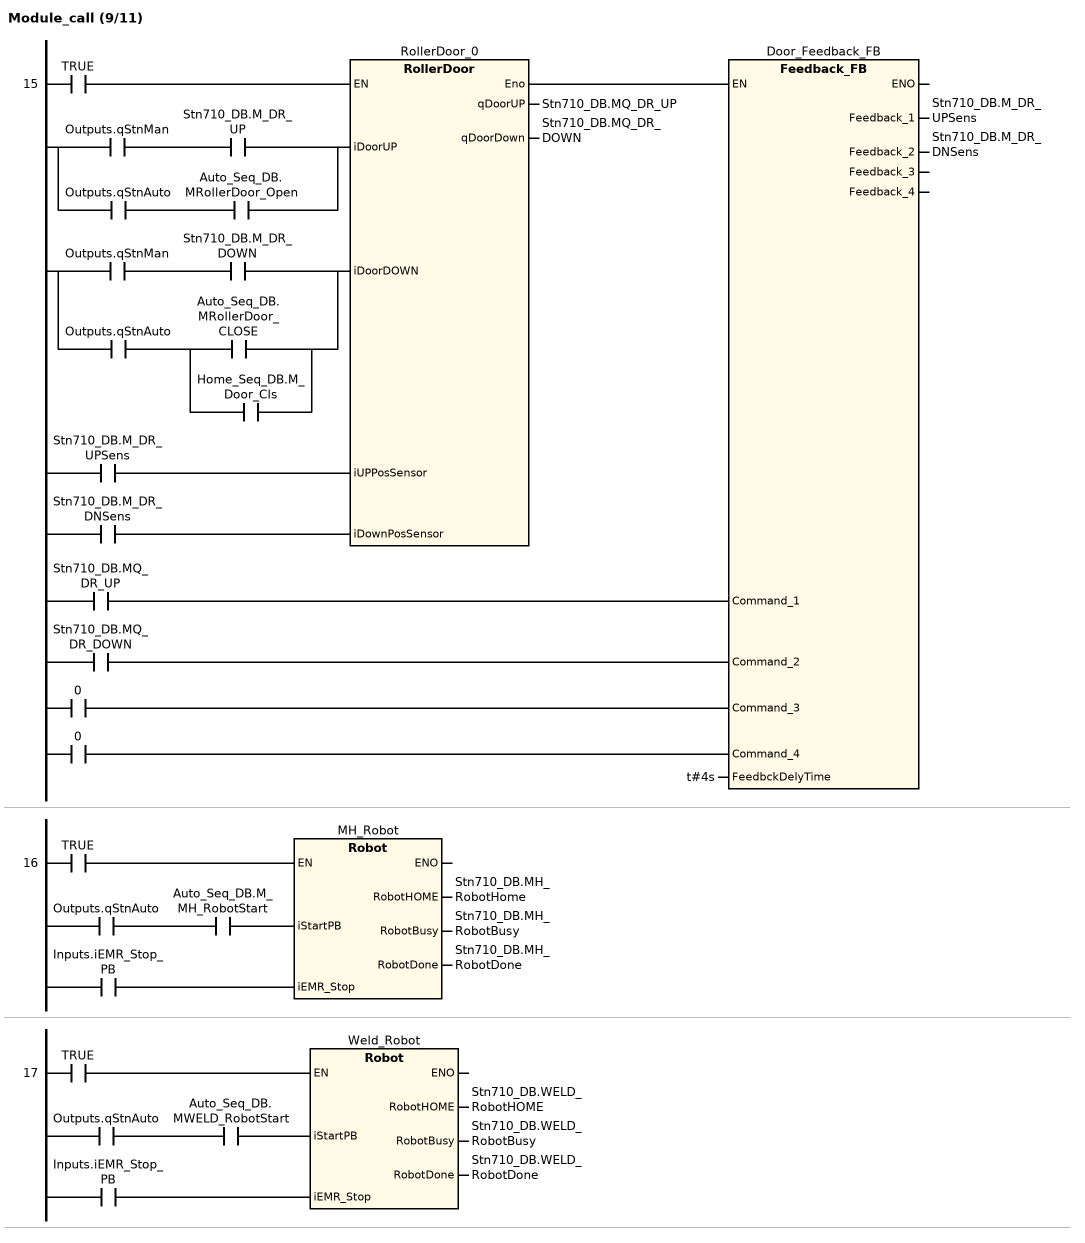
// NETWORK 15
RollerDoor_0(
    EN := TRUE,
    iDoorUP := Outputs.qStnMan AND Stn710_DB.M_DR_UP OR Outputs.qStnAuto AND Auto_Seq_DB.MRollerDoor_Open,
    iDoorDOWN := Outputs.qStnMan AND Stn710_DB.M_DR_DOWN OR Outputs.qStnAuto AND (Auto_Seq_DB.MRollerDoor_CLOSE OR Home_Seq_DB.M_Door_Cls),
    iUPPosSensor := Stn710_DB.M_DR_UPSens,
    iDownPosSensor := Stn710_DB.M_DR_DNSens,
    qDoorUP => Stn710_DB.MQ_DR_UP,
    qDoorDown => Stn710_DB.MQ_DR_DOWN); // RollerDoor
Door_Feedback_FB(
    EN := TRUE,
    Command_1 := Stn710_DB.MQ_DR_UP,
    Command_2 := Stn710_DB.MQ_DR_DOWN,
    Command_3 := 0,
    Command_4 := 0,
    FeedbckDelyTime := t#4s,
    Feedback_1 => Stn710_DB.M_DR_UPSens,
    Feedback_2 => Stn710_DB.M_DR_DNSens); // Feedback_FB

// NETWORK 16
MH_Robot(
    EN := TRUE,
    iStartPB := Outputs.qStnAuto AND Auto_Seq_DB.M_MH_RobotStart,
    iEMR_Stop := Inputs.iEMR_Stop_PB,
    RobotHOME => Stn710_DB.MH_RobotHome,
    RobotBusy => Stn710_DB.MH_RobotBusy,
    RobotDone => Stn710_DB.MH_RobotDone); // Robot

// NETWORK 17
Weld_Robot(
    EN := TRUE,
    iStartPB := Outputs.qStnAuto AND Auto_Seq_DB.MWELD_RobotStart,
    iEMR_Stop := Inputs.iEMR_Stop_PB,
    RobotHOME => Stn710_DB.WELD_RobotHOME,
    RobotBusy => Stn710_DB.WELD_RobotBusy,
    RobotDone => Stn710_DB.WELD_RobotDone); // Robot

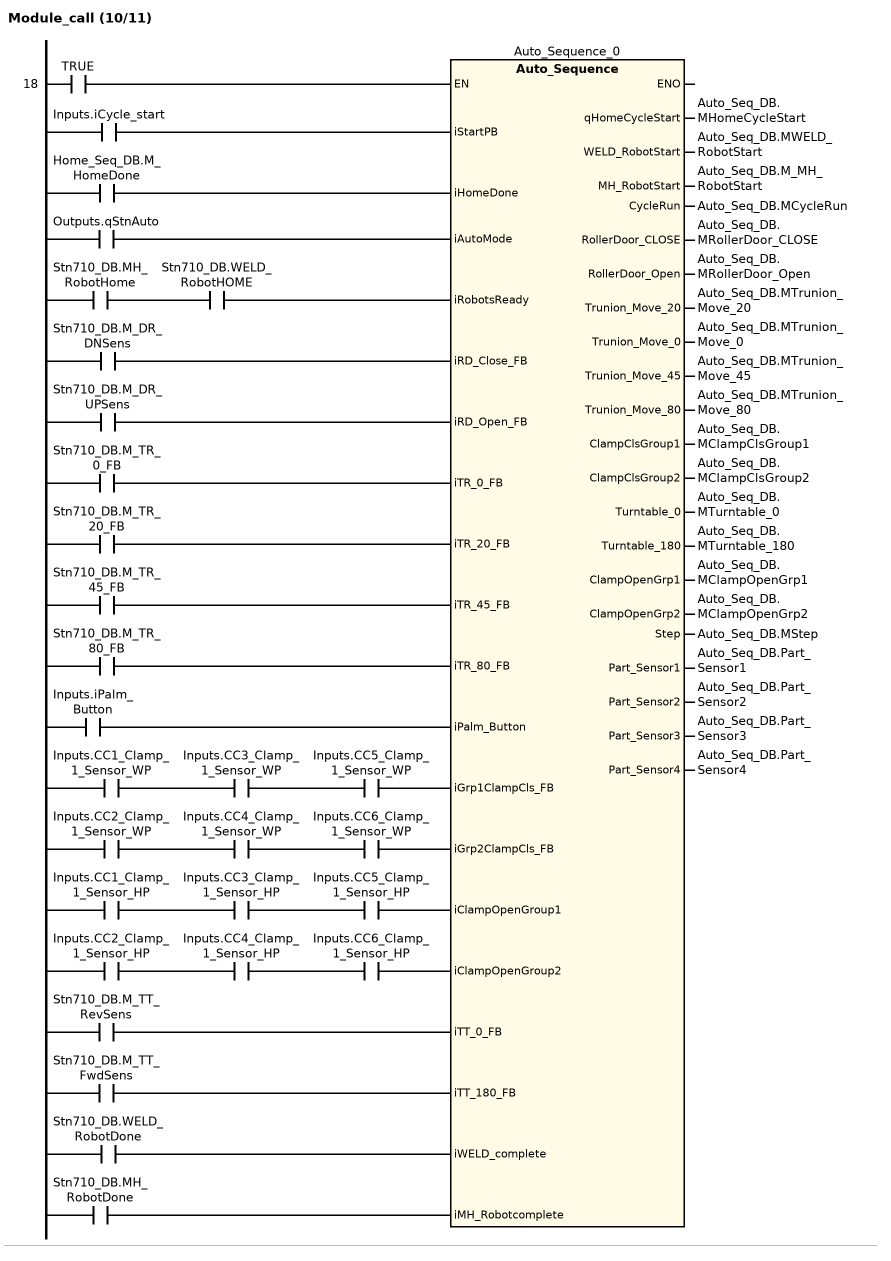
// NETWORK 18
Auto_Sequence_0(
    EN := TRUE,
    iStartPB := Inputs.iCycle_start,
    iHomeDone := Home_Seq_DB.M_HomeDone,
    iAutoMode := Outputs.qStnAuto,
    iRobotsReady := Stn710_DB.MH_RobotHome AND Stn710_DB.WELD_RobotHOME,
    iRD_Close_FB := Stn710_DB.M_DR_DNSens,
    iRD_Open_FB := Stn710_DB.M_DR_UPSens,
    iTR_0_FB := Stn710_DB.M_TR_0_FB,
    iTR_20_FB := Stn710_DB.M_TR_20_FB,
    iTR_45_FB := Stn710_DB.M_TR_45_FB,
    iTR_80_FB := Stn710_DB.M_TR_80_FB,
    iPalm_Button := Inputs.iPalm_Button,
    iGrp1ClampCls_FB := Inputs.CC1_Clamp_1_Sensor_WP AND Inputs.CC3_Clamp_1_Sensor_WP AND Inputs.CC5_Clamp_1_Sensor_WP,
    iGrp2ClampCls_FB := Inputs.CC2_Clamp_1_Sensor_WP AND Inputs.CC4_Clamp_1_Sensor_WP AND Inputs.CC6_Clamp_1_Sensor_WP,
    iClampOpenGroup1 := Inputs.CC1_Clamp_1_Sensor_HP AND Inputs.CC3_Clamp_1_Sensor_HP AND Inputs.CC5_Clamp_1_Sensor_HP,
    iClampOpenGroup2 := Inputs.CC2_Clamp_1_Sensor_HP AND Inputs.CC4_Clamp_1_Sensor_HP AND Inputs.CC6_Clamp_1_Sensor_HP,
    iTT_0_FB := Stn710_DB.M_TT_RevSens,
    iTT_180_FB := Stn710_DB.M_TT_FwdSens,
    iWELD_complete := Stn710_DB.WELD_RobotDone,
    iMH_Robotcomplete := Stn710_DB.MH_RobotDone,
    qHomeCycleStart => Auto_Seq_DB.MHomeCycleStart,
    WELD_RobotStart => Auto_Seq_DB.MWELD_RobotStart,
    MH_RobotStart => Auto_Seq_DB.M_MH_RobotStart,
    CycleRun => Auto_Seq_DB.MCycleRun,
    RollerDoor_CLOSE => Auto_Seq_DB.MRollerDoor_CLOSE,
    RollerDoor_Open => Auto_Seq_DB.MRollerDoor_Open,
    Trunion_Move_20 => Auto_Seq_DB.MTrunion_Move_20,
    Trunion_Move_0 => Auto_Seq_DB.MTrunion_Move_0,
    Trunion_Move_45 => Auto_Seq_DB.MTrunion_Move_45,
    Trunion_Move_80 => Auto_Seq_DB.MTrunion_Move_80,
    ClampClsGroup1 => Auto_Seq_DB.MClampClsGroup1,
    ClampClsGroup2 => Auto_Seq_DB.MClampClsGroup2,
    Turntable_0 => Auto_Seq_DB.MTurntable_0,
    Turntable_180 => Auto_Seq_DB.MTurntable_180,
    ClampOpenGrp1 => Auto_Seq_DB.MClampOpenGrp1,
    ClampOpenGrp2 => Auto_Seq_DB.MClampOpenGrp2,
    Step => Auto_Seq_DB.MStep,
    Part_Sensor1 => Auto_Seq_DB.Part_Sensor1,
    Part_Sensor2 => Auto_Seq_DB.Part_Sensor2,
    Part_Sensor3 => Auto_Seq_DB.Part_Sensor3,
    Part_Sensor4 => Auto_Seq_DB.Part_Sensor4); // Auto_Sequence

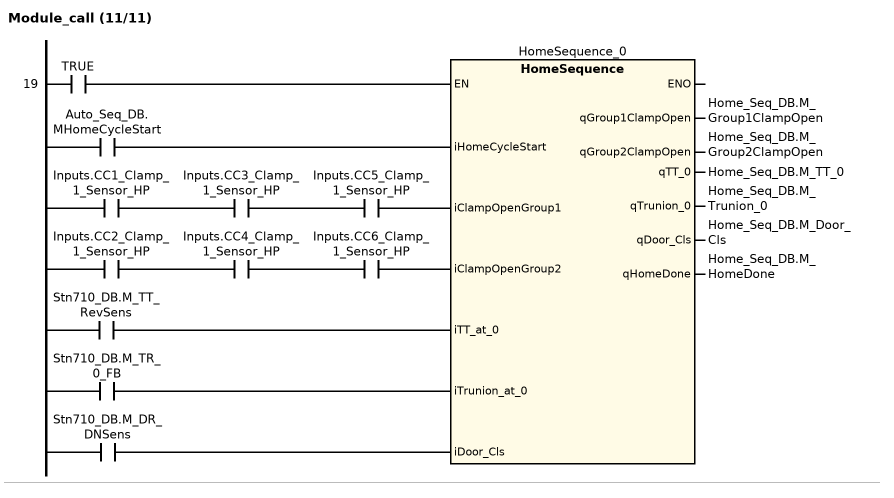
// NETWORK 19
HomeSequence_0(
    EN := TRUE,
    iHomeCycleStart := Auto_Seq_DB.MHomeCycleStart,
    iClampOpenGroup1 := Inputs.CC1_Clamp_1_Sensor_HP AND Inputs.CC3_Clamp_1_Sensor_HP AND Inputs.CC5_Clamp_1_Sensor_HP,
    iClampOpenGroup2 := Inputs.CC2_Clamp_1_Sensor_HP AND Inputs.CC4_Clamp_1_Sensor_HP AND Inputs.CC6_Clamp_1_Sensor_HP,
    iTT_at_0 := Stn710_DB.M_TT_RevSens,
    iTrunion_at_0 := Stn710_DB.M_TR_0_FB,
    iDoor_Cls := Stn710_DB.M_DR_DNSens,
    qGroup1ClampOpen => Home_Seq_DB.M_Group1ClampOpen,
    qGroup2ClampOpen => Home_Seq_DB.M_Group2ClampOpen,
    qTT_0 => Home_Seq_DB.M_TT_0,
    qTrunion_0 => Home_Seq_DB.M_Trunion_0,
    qDoor_Cls => Home_Seq_DB.M_Door_Cls,
    qHomeDone => Home_Seq_DB.M_HomeDone); // HomeSequence

END_FUNCTION_BLOCK

// ---- POUs/Library/FB_CylinderModule.TcPOU
FUNCTION_BLOCK FB_CylinderModule
VAR_INPUT
    iResetFaults:BOOL;//Reset Fault CMD
    iWorkCmd:BOOL ;//Cyl Work Postion CMD
    iHomeCmd:BOOL ;//Cyl Home Postion CMD
    iWorkSen:BOOL ;// Cyl Work Postion Input
    iHomeSen:BOOL ;// Cyl Home Postion Input
    iWorkCleartoMove:BOOL ;// Condition Healthy then 1
    iHomeCleartoMove:BOOL ;// Condition Healthy then 1
    iTimeoutValue:TIME ;// Time Required E.gT#500MS,T#2S
END_VAR
VAR_OUTPUT
	qENO   : BOOL; //  Block Enable
	qWorkSol    : BOOL; // Cyl Work Position Sol Output
    qHomeSol: BOOL; //Cyl Home Position Sol Output
    qWorkOver: BOOL; // Cyl AT Work Position
    qHomeOver: BOOL; //Cyl AT Home Position
    qErrHomeInterlock: BOOL; //homeCleartoMove is low AND home command is active.
    qErrHomeTout: BOOL; //cylinder did NOT reachhome position within definedTIME
    qErrWorkInterlock: BOOL; //WorkCleartoMove is low AND work command is active.
    qErrWorkTout: BOOL; //cylinder did NOT reachwork position within definedtime
END_VAR
VAR
	sFltRstPls: BOOL; //Stat BIT FOR positive edge OF reset fault input
    sFltEdge: R_TRIG; //Positive edge OF fault reset input
    sTimeoutValue: TIME; //Stat BIT FOR TIME out value
    sHomeSol: BOOL; //
    sWorkSol: BOOL; //
    sErrWorkInterlock: BOOL; 
    sErrHomeInterlock: BOOL; 
    sErrWorkTout: BOOL; 
    sErrHomeTOut: BOOL; 
    sWorkOver: BOOL; 
    sHomeOver: BOOL; 
    sErrWorkCommon: BOOL; 
    sErrHomeCommon: BOOL; 
	sDlyTimeOutt: TON;
END_VAR

 // Rising Edge Detection for Fault Reset
sFltEdge(CLK := iResetFaults);
sFltRstPls := sFltEdge.Q;

 // Work Command Logic
IF (
    (iWorkCmd AND iWorkCleartomove) OR 
    (sWorkSol AND iWorkSen AND NOT iHomeSen)
   )
   AND NOT iHomeCmd
   AND NOT sHomeSol
THEN
    sWorkSol := TRUE;
ELSE
    sWorkSol := FALSE;
END_IF;
// Home Command Logic
IF (
    (iHomeCmd AND iHomeCleartomove) OR 
    (sHomeSol AND iHomeSen AND NOT iWorkSen)
   )
   AND NOT iWorkCmd
   AND NOT sWorkSol
THEN
    sHomeSol := TRUE;
ELSE
    sHomeSol := FALSE;
END_IF;
// Work Interlock Error
IF (iWorkCmd AND NOT iWorkCleartomove) THEN
    sErrWorkInterlock := TRUE;
ELSIF (sFltRstPls) THEN
    sErrWorkInterlock := FALSE;
END_IF;
// Home Interlock Error
IF (iHomeCmd AND NOT iHomeCleartomove) THEN
    sErrHomeInterlock := TRUE;
ELSIF (sFltRstPls) THEN
    sErrHomeInterlock := FALSE;
END_IF;
// Sensor Timeout Timer
sDlyTimeOutt(
    IN := (
            (sWorkSol AND NOT iWorkSen AND NOT sErrWorkTout)
         OR (sHomeSol AND NOT iHomeSen AND NOT sErrHomeTout)
          ),
    PT := iTimeoutValue
);
//sDlyTimeOutt.Q:= sDlyTimeOutt.Q;
//Work Timeout Error
IF (
   (sWorkSol AND NOT iWorkSen AND sDlyTimeOutt.Q) OR
   (sErrWorkTout AND NOT sFltRstPls)
   )
   THEN
   sErrWorkTout := TRUE;
   ELSE
	   sErrWorkTout := FALSE;
   END_IF;
   
   //Home Timeout Error
IF (
   (sHomeSol AND NOT iHomeSen AND sDlyTimeOutt.Q) OR
   (sErrHomeTOut AND NOT sFltRstPls)
   )
   THEN
   sErrHomeTOut := TRUE;
   ELSE
	   sErrHomeTOut := FALSE;
   END_IF;
	
//Workover
IF (
   (iWorkSen AND NOT iHomeSen ) 
   )
   THEN
   sWorkOver := TRUE;
   ELSE
	   sWorkOver := FALSE;
   END_IF; 
//Homeover
IF (
   (iHomeSen AND NOT iWorkSen) 
   )
   THEN
   sHomeOver := TRUE;
   ELSE
	   sHomeOver := FALSE;
   END_IF;   
   
   qHomeSol := sHomeSol;
   qWorkSol := sWorkSol;
   qErrWorkinterlock := sErrWorkinterlock;
   qErrHomeinterlock := sErrHomeinterlock;
   qErrWorkTout := sErrWorkTout;
   qErrHomeTout := sErrHomeTOut;
   qWorkOver := sWorkOver;
   qHomeOver := sHomeOver;

END_FUNCTION_BLOCK

// ---- POUs/Library/Feedback_FB.TcPOU
FUNCTION_BLOCK Feedback_FB
VAR_INPUT
	EN : BOOL;
	Command_1  : BOOL;
	Command_2  : BOOL;
	Command_3  : BOOL;
	Command_4  : BOOL;
	FeedbckDelyTime  : TIME;
END_VAR
VAR_OUTPUT
	ENO           : BOOL;
	Feedback_1    : BOOL;     
    Feedback_2    : BOOL;
	Feedback_3    : BOOL;     
    Feedback_4    : BOOL;
END_VAR
VAR
	fb1_Time       : TON;
	fb2_Time       : TON;
	fb3_Time       : TON;
	fb4_Time       : TON;
END_VAR

//FEEDBACK 1 DELAY

IF Command_1 THEN
	fb1_Time(IN := Command_1, PT :=FeedbckDelyTime);
	Feedback_1 := fb1_Time.Q;
	Feedback_2 := FALSE;
	Feedback_3 := FALSE;
	Feedback_4 := FALSE;
ELSE 
	fb1_Time(IN := FALSE);
END_IF;
	
//FEEDBACK 2 DELAY

IF Command_2 THEN
	fb2_Time(IN := Command_2, PT := FeedbckDelyTime);
	Feedback_2 := fb2_Time.Q;
	Feedback_1 := FALSE;
	Feedback_3 := FALSE;
	Feedback_4 := FALSE;
ELSE 
	fb2_Time(IN := FALSE);
END_IF;

//FEEDBACK 3 DELAY

IF Command_3 THEN
	fb3_Time(IN := Command_3, PT :=FeedbckDelyTime);
	Feedback_3 := fb3_Time.Q;
	Feedback_1 := FALSE;
	Feedback_2 := FALSE;
	Feedback_4 := FALSE;
ELSE 
	fb3_Time(IN := FALSE);
END_IF;
	
//FEEDBACK 4 DELAY

IF Command_4 THEN
	fb4_Time(IN := Command_4, PT := FeedbckDelyTime);
	Feedback_4 := fb4_Time.Q;
	Feedback_1 := FALSE;
	Feedback_2 := FALSE;
	Feedback_3 := FALSE;
ELSE 
	fb4_Time(IN := FALSE);
END_IF;

END_FUNCTION_BLOCK

// ---- POUs/PowerOn.TcPOU
FUNCTION_BLOCK PowerOn
VAR_INPUT
	iControl_on  	: BOOL;
	iControl_off    : BOOL;
	iAuto_Man 		: BOOL;
	iEMRSTOP		: bool;
END_VAR
VAR_OUTPUT
	 ENO    : BOOL;
	qPower_On	 : BOOL;
	qStnAuto	 :BOOL;
	qStnMan  	 : BOOL;
END_VAR
VAR	
END_VAR

// Control ON Logic
IF iControl_On AND NOT iControl_off AND (Stn710_DB.Alarm_count = 0 OR Stn710_DB.Alarm_count > 1)  THEN
	qPower_On := TRUE;	
	ELSE
	qPower_On := FALSE;
END_IF

// Auto Logic
IF qPower_On AND NOT iAuto_Man THEN
	qStnAuto := TRUE;
	qStnMan := FALSE;
	ELSE
	qStnAuto := FALSE;	
END_IF
// Manual Logic
IF qPower_On AND iAuto_Man THEN
	qStnMan := TRUE;
	qStnAuto := FALSE;
	
	ELSE
	qStnMan := FALSE;	
END_IF

END_FUNCTION_BLOCK

// ---- POUs/TurnTable.TcPOU
FUNCTION_BLOCK TurnTable
VAR_INPUT
	EN   : BOOL;
	iStartCW    	:  BOOL;    // Clockwise Move Command 
	iStartCCW   	:  BOOL;    // Counterclockwise Move Command 
	iFwdPosSensor  	:  BOOL;    // Forward Position sensor 180* feedback
	iRevPosSensor  	:  BOOL;    // Forward Position sensor 0* feedback
END_VAR
VAR_OUTPUT
	Eno  : BOOL;
	qMotorRun  :  BOOL ; 	// Motor Run Status
	qMotorDir  :  BOOL ;    // Motor Direction Status 
END_VAR
VAR
END_VAR

// Motor Safety
IF  iStartCW AND iStartCCW THEN
	qMotorRun := FALSE;
	qMotorDir := FALSE;
END_IF

// TURNTABLE OPERATION
	IF iStartCW AND NOT iFwdPosSensor THEN
		qMotorRun := TRUE;
		qMotorDir := FALSE;
	ELSIF iStartCCW AND NOT iRevPosSensor THEN
		qMotorRun := TRUE;
		qMotorDir := TRUE;
		ELSE 
		qMotorRun := FALSE;
		qMotorDir := FALSE;
	END_IF

END_FUNCTION_BLOCK

// ---- POUs/Trunion.TcPOU
FUNCTION_BLOCK Trunion
VAR_INPUT
	EN   : BOOL;
	iStart0    		:  BOOL;    // Clockwise Move Command 
	iStart20   		:  BOOL;    // Counterclockwise Move Command 
	iStart45    	:  BOOL;    // Clockwise Move Command 
	iStart80   		:  BOOL;    // Counterclockwise Move Command 
	i0PosSensor  	:  BOOL;    // Forward Position sensor 180* feedback
	i20PosSensor  	:  BOOL;    // Forward Position sensor 0* feedback
	i45PosSensor  	:  BOOL;    // Forward Position sensor 180* feedback
	i80PosSensor  	:  BOOL;    // Forward Position sensor 0* feedback
END_VAR
VAR_OUTPUT
	Eno  : BOOL;
	qMotor0 	 :  BOOL ; 	// Motor Run Status
	qMotor20  	:  BOOL ;    // Motor Direction Status 
	qMotor45 	 :  BOOL ; 	// Motor Run Status
	qMotor80  	:  BOOL ;    // Motor Direction Status 
END_VAR
VAR
END_VAR

// TRUNION OPERATION
IF iStart0 AND NOT i0PosSensor THEN
		qMotor0  := TRUE;
	ELSIF iStart20 AND NOT i20PosSensor THEN
		qMotor20 := TRUE;
	ELSIF iStart45 AND NOT i45PosSensor THEN
		qMotor45 := TRUE;
	ELSIF iStart80 AND NOT i80PosSensor THEN
		qMotor80 := TRUE;
	ELSE qMotor0 := FALSE;
		 qMotor20 := FALSE;
		 qMotor45 := FALSE;
		 qMotor80 := FALSE;
	END_IF

END_FUNCTION_BLOCK

// ---- POUs/RollerDoor.TcPOU
FUNCTION_BLOCK PUBLIC RollerDoor
VAR_INPUT
	EN   : BOOL;
	iDoorUP    		:  BOOL;    // Clockwise Move Command 
	iDoorDOWN   	:  BOOL;    // Counterclockwise Move Command 
	iUPPosSensor  	:  BOOL;    // Forward Position sensor 180* feedback
	iDownPosSensor  :  BOOL;    // Forward Position sensor 0* feedback
END_VAR
VAR_OUTPUT
	Eno  : BOOL;
	qDoorUP		 	:  BOOL ; 	// Motor Run Status
	qDoorDown	  	:  BOOL ;    // Motor Direction Status 
END_VAR
VAR
END_VAR

// Door Safety
IF  iDoorUP AND iDoorDOWN THEN
	qDoorUP 	:= FALSE;
	qDoorDown 	:= FALSE;
END_IF

//DOOR operation
	IF iDoorUP AND NOT iUPPosSensor THEN
		qDoorUP := TRUE;
	ELSIF iDoorDOWN AND NOT iDownPosSensor THEN
		qDoorDown := TRUE;
	ELSE 
		qDoorUP := FALSE;
		qDoorDOWN := FALSE;
	END_IF

END_FUNCTION_BLOCK

// ---- POUs/Robot.TcPOU
FUNCTION_BLOCK Robot
VAR_INPUT
	EN				:BOOL;
	iStartPB		:BOOL;
	iEMR_Stop		:BOOL;
END_VAR
VAR_OUTPUT
	ENO				: BOOL;
	RobotHOME		: BOOL;
	RobotBusy		:BOOL;
	RobotDone		:BOOL;
END_VAR
VAR
	MH_Time		:TON;
	StepNo		:INT;
	MHProgramNo	:INT;
	RobotStart	:BOOL;	
END_VAR

IF iEMR_Stop THEN 
StepNo := 0;	
END_IF

CASE StepNo OF
0:   RobotHOME := TRUE;
     RobotBusy := FALSE;
	 MH_Time(IN :=FALSE);
	 RobotDone := FALSE;
    IF iStartPB AND NOT iEMR_Stop THEN
       StepNo := 10;
    END_IF;

10:
    MHProgramNo := 1;
	RobotBusy := TRUE;
	RobotHOME := FALSE;
    StepNo := 20;

20:
	MH_Time(IN := TRUE, PT :=T#5S);
   IF MH_Time.Q THEN
		RobotDone := TRUE; 
		RobotStart := FALSE; 
		RobotBusy := FALSE;
		StepNo := 30;
    END_IF;

30:
    IF RobotDone THEN
       StepNo := 0;
    END_IF;

END_CASE;

END_FUNCTION_BLOCK

// ---- POUs/Auto_Sequence.TcPOU
FUNCTION_BLOCK Auto_Sequence
VAR_INPUT
	EN				:BOOL;
	iStartPB		:BOOL;
	iHomeDone		:BOOL;
	iAutoMode		:BOOL;
	iRobotsReady	:BOOL;
	iRD_Close_FB	:BOOL;
	iRD_Open_FB		:BOOL;
	iTR_0_FB		:BOOL;
	iTR_20_FB		:BOOL;
	iTR_45_FB		:BOOL;
	iTR_80_FB		:BOOL;
	iPalm_Button	:BOOL;
	iGrp1ClampCls_FB :BOOL;
	iGrp2ClampCls_FB :BOOL;
	iClampOpenGroup1 :BOOL;
	iClampOpenGroup2 :BOOL;
	iTT_0_FB		:BOOL;
	iTT_180_FB		:BOOL;
	iWELD_complete	:BOOL;
	iMH_Robotcomplete	:BOOL;

END_VAR
VAR_OUTPUT
	ENO					:BOOL;
	qHomeCycleStart 	:BOOL;
	WELD_RobotStart		:BOOL;
	MH_RobotStart		:BOOL;
	CycleRun			:BOOL;
	RollerDoor_CLOSE	:BOOL;
	RollerDoor_Open		:BOOL;
	Trunion_Move_20		:BOOL;
	Trunion_Move_0		:BOOL;
	Trunion_Move_45		:BOOL;
	Trunion_Move_80		:BOOL;
	ClampClsGroup1		:BOOL;
	ClampClsGroup2		:BOOL;
	Turntable_0			:BOOL;
	Turntable_180		:BOOL;
	ClampOpenGrp1		:BOOL;
	ClampOpenGrp2		:BOOL;
	Step				:INT;
	Part_Sensor1		:BOOL;
	Part_Sensor2		:BOOL;
	Part_Sensor3		:BOOL;
	Part_Sensor4		:BOOL;
END_VAR
VAR
	StartPulse		: R_TRIG;
	StepNo			: INT;
	RD_CLOSE1		:BOOL;
	RD_CLOSE2		:BOOL;
	RD_CLOSE3		:BOOL;
	RD_OPEN1		:BOOL;
	RD_OPEN2		:BOOL;
	RD_OPEN3		:BOOL;
END_VAR

    StartPulse(CLK := iStartPB);
	RollerDoor_CLOSE := RD_CLOSE1 OR RD_CLOSE2 OR RD_CLOSE3;
	RollerDoor_Open := RD_OPEN1 OR RD_OPEN2 OR RD_OPEN3;
	Step := StepNo;
	
	
// Step reset logic
IF NOT iAutoMode THEN
	StepNo := 0;
	RD_CLOSE1 := FALSE;
	WELD_RobotStart := FALSE;
	MH_RobotStart := FALSE;
	qHomeCycleStart := FALSE;
	Trunion_Move_20:=FALSE;
	RD_OPEN1 := FALSE;
	Trunion_Move_80 := FALSE;
	RD_OPEN2 := FALSE;
	RD_CLOSE3 := FALSE;
	Turntable_180 := FALSE;
	Trunion_Move_0:= FALSE;
	ClampClsGroup1 := FALSE;
	ClampClsGroup2 := FALSE;
	RD_OPEN3 := FALSE;
	Trunion_Move_45 := FALSE;
END_IF


IF iAutoMode THEN 

    StartPulse(CLK := iStartPB);
	
    CASE StepNo OF
// CYCLE START

    0:
        WELD_RobotStart := FALSE;
		MH_RobotStart := FALSE;

        IF  iStartPB AND iRobotsReady THEN
			StepNo := 5;
        END_IF;
		
// Call Home Cycle

    5:
      qHomeCycleStart := TRUE;

        IF iHomeDone THEN
			qHomeCycleStart := FALSE;
            StepNo := 10;
        END_IF;
		
// RD_CLOSE

    10:
        RD_CLOSE1 := TRUE;

        IF iRD_Close_FB THEN
			RD_CLOSE1 := FALSE;
            StepNo := 20;
        END_IF;
		
// TRUNION

    20:
        Trunion_Move_20 := TRUE;

        IF iTR_20_FB THEN
			Trunion_Move_20:=FALSE;
            StepNo := 30;
        END_IF;
		
// RD_OPEN

    30:
        RD_OPEN1 := TRUE;

        IF iRD_Open_FB THEN
            StepNo := 40;
			RD_OPEN1 := FALSE;
        END_IF;

// Operator Load_1ST PART

    40:
         Part_Sensor1 := TRUE;
	   IF  Part_Sensor1 AND iPalm_Button THEN
            StepNo := 50;
        END_IF;

// Operator Load_2ND PART

     50:
		Part_Sensor2 := TRUE;
	   IF Part_Sensor2 AND iPalm_Button THEN
            StepNo := 60;
        END_IF;
		
// Clamp Close_1ST,3RD,5TH

    60:
        ClampClsGroup1 := TRUE;
        IF iGrp1ClampCls_FB THEN
            StepNo := 70;
        END_IF;
		
// RD_CLOSE

    70:
        RD_CLOSE2 := TRUE;
    	ClampClsGroup1 := FALSE;
        IF iGrp1ClampCls_FB AND iRD_Close_FB THEN
            StepNo := 80;
        END_IF;

// TRUNION


    80:
        Trunion_Move_80 := TRUE;
        RD_CLOSE2 := FALSE;
        IF iTR_80_FB THEN
			Trunion_Move_80 := FALSE;
            StepNo := 90;
        END_IF;

// RD_OPEN-0


    90:
        RD_OPEN2 := TRUE;
       IF iRD_Open_FB THEN
			RD_OPEN2 := FALSE;
            StepNo := 100;
        END_IF;

// Operator Load_3RD_PART

    100:
       Part_Sensor3 := TRUE ;
	   IF Part_Sensor3 AND iPalm_Button THEN
            StepNo := 110;
        END_IF;

// Operator Load_4TH_PART

    110:
		Part_Sensor4 := TRUE;
	   IF Part_Sensor4 AND iPalm_Button THEN
            StepNo := 120;
        END_IF;

// RD_CLOSE-0

    120:
        RD_CLOSE3 := TRUE;
        IF iRD_Close_FB THEN
			RD_CLOSE3 := FALSE;
            StepNo := 130;
        END_IF;

//  CLAMP CLOSE 2ND,4TH, 6TH


    130:
	 ClampClsGroup2 := TRUE;
	 IF iGrp2ClampCls_FB THEN
		StepNo := 140;
        END_IF;

// TURNTABLE-180* AND TRUNION_0*


    140: 
		ClampClsGroup2 := FALSE;
		Trunion_Move_0:= TRUE;
		Turntable_180 := TRUE;
		
		IF iTT_180_FB AND iTR_0_FB THEN
			Turntable_180 := FALSE;
			Trunion_Move_0:= FALSE;
			StepNo := 150;
		END_IF;
   
// Start WELD_Robot

    150:
        WELD_RobotStart := TRUE;

        IF iWELD_complete THEN
            WELD_RobotStart := FALSE;
            StepNo := 160;
        END_IF;

// CLAMP OPEN 1ST,3RD,5TH

    160:
        CycleRun := TRUE;
		ClampOpenGrp1 := TRUE;
        IF  iClampOpenGroup1 THEN
	    ClampOpenGrp1 := FALSE;
		StepNo := 170;
        END_IF;

// RD_OPEN
	
	170: 
        RD_OPEN3 := TRUE;
        
        IF RollerDoor_Open THEN
			RD_OPEN3 := FALSE;
            StepNo := 180;
        END_IF;

// Start MH_Robot_1ST

    180:
        MH_RobotStart := TRUE;
		Part_Sensor1 := FALSE;
        Part_Sensor2 := FALSE;
        IF iMH_Robotcomplete AND NOT Part_Sensor1 AND NOT Part_Sensor2  THEN
            MH_RobotStart := FALSE;
            StepNo := 190;
        END_IF;

// TRUNION_45

	 190:
        Trunion_Move_45 := TRUE;
     	RD_CLOSE3 := FALSE;
        IF iTR_45_FB THEN
			Trunion_Move_45 := FALSE;
            StepNo := 200;
        END_IF;
    
// Start UNCLAMP 2ND, 4TH,6TH
		
    200:
        CycleRun := TRUE;
		ClampOpenGrp2 := TRUE;
        IF iClampOpenGroup2 THEN
	    ClampOpenGrp2 := FALSE;
            StepNo := 210;
        END_IF;

// Start MH_Robot_2ND

		
     210:
        MH_RobotStart := TRUE;
		Part_Sensor3 := FALSE;
		Part_Sensor4 := FALSE;
        IF iMH_Robotcomplete AND NOT Part_Sensor3 AND NOT Part_Sensor4 THEN
            MH_RobotStart := FALSE;
            StepNo := 220;
        END_IF;
// -----------------------------------
    // Cycle Finish
    // -----------------------------------

    220:
        CycleRun := FALSE;
        
        StepNo := 0;

    END_CASE;

END_IF;

END_FUNCTION_BLOCK

// ---- POUs/HomeSequence.TcPOU
FUNCTION_BLOCK HomeSequence
VAR_INPUT
	EN :BOOL;
	iHomeCycleStart :BOOL;
	iClampOpenGroup1 :BOOL;
	iClampOpenGroup2 :BOOL;
	iTT_at_0 : BOOL;
	iTrunion_at_0 :BOOL;
	iDoor_Cls : BOOL;
END_VAR
VAR_OUTPUT
	ENO :BOOL;
	qGroup1ClampOpen :BOOL;
	qGroup2ClampOpen :BOOL;
	qTT_0 : BOOL;
	qTrunion_0 : BOOL;
	qDoor_Cls : BOOL;
	qHomeDone : BOOL;
END_VAR
VAR
	StepNo : INT;
END_VAR

CASE StepNo OF
	
0:
	qHomeDone := FALSE;
	IF iHomeCycleStart THEN
	StepNo := 10;
	END_IF

// All Clamps home
10:
	qGroup1ClampOpen := TRUE;
	qGroup2ClampOpen := TRUE;
	IF iClampOpenGroup1 AND iClampOpenGroup2 THEN
		qGroup1ClampOpen := FALSE;
		qGroup2ClampOpen := FALSE;
		StepNo := 20;
	END_IF

// Roller door close
20:
	qDoor_Cls := TRUE;
	IF iDoor_Cls THEN
		qDoor_Cls := FALSE;
		StepNo := 30;
	END_IF
	
// Trunion to 0* position
30:
	qTrunion_0 := TRUE;
	IF iTrunion_at_0 THEN
		qTrunion_0 := FALSE;
		StepNo := 40;
	END_IF

// Turn Table to home position
40:
	qTT_0 := TRUE;
	IF iTT_at_0 THEN
		qTT_0 := FALSE;
		qHomeDone := TRUE;
		StepNo := 0;
	END_IF
	
END_CASE

END_FUNCTION_BLOCK

// ---- POUs/Alarms.TcPOU
FUNCTION_BLOCK Alarms
VAR_INPUT
	EN : BOOL;
END_VAR
VAR_OUTPUT
		ENO : BOOL;
END_VAR
VAR
END_VAR

//Reset All Alarms
IF Inputs.iResetFault THEN
	Alarm_DB.EMR_Stop_pressed := FALSE;
	Stn710_DB.Alarm_count := 0;
END_IF

//EMERGENCY STOP ALARM
IF Inputs.iEMR_Stop_PB THEN
	Alarm_DB.EMR_Stop_pressed := TRUE;
	Stn710_DB.Alarm_count := 1;
END_IF

IF Stn710_DB.CC1_CLAMP.ErrHomeInterlock THEN
	Stn710_DB.Alarm_count := 2;
END_IF

IF Stn710_DB.CC1_CLAMP.ErrHomeTout THEN
	Stn710_DB.Alarm_count := 3;
END_IF

IF Stn710_DB.CC1_CLAMP.ErrWorkInterlock THEN
	Stn710_DB.Alarm_count := 4;
END_IF

IF Stn710_DB.CC1_CLAMP.ErrWorkTout THEN
	Stn710_DB.Alarm_count := 5;
END_IF

IF Stn710_DB.CC2_CLAMP.ErrHomeInterlock THEN
	Stn710_DB.Alarm_count := 6;
END_IF

IF Stn710_DB.CC2_CLAMP.ErrHomeTout THEN
	Stn710_DB.Alarm_count := 7;
END_IF

IF Stn710_DB.CC2_CLAMP.ErrWorkInterlock THEN
	Stn710_DB.Alarm_count := 8;
END_IF

IF Stn710_DB.CC2_CLAMP.ErrWorkTout THEN
	Stn710_DB.Alarm_count := 9;
END_IF

IF Stn710_DB.CC3_CLAMP.ErrHomeInterlock THEN
	Stn710_DB.Alarm_count := 10;
END_IF

IF Stn710_DB.CC3_CLAMP.ErrHomeTout THEN
	Stn710_DB.Alarm_count := 11;
END_IF

IF Stn710_DB.CC3_CLAMP.ErrWorkInterlock THEN
	Stn710_DB.Alarm_count := 12;
END_IF

IF Stn710_DB.CC3_CLAMP.ErrWorkTout THEN
	Stn710_DB.Alarm_count := 13;
END_IF

IF Stn710_DB.CC4_CLAMP.ErrHomeInterlock THEN
	Stn710_DB.Alarm_count := 14;
END_IF

IF Stn710_DB.CC4_CLAMP.ErrHomeTout THEN
	Stn710_DB.Alarm_count := 15;
END_IF

IF Stn710_DB.CC4_CLAMP.ErrWorkInterlock THEN
	Stn710_DB.Alarm_count := 16;
END_IF

IF Stn710_DB.CC4_CLAMP.ErrWorkTout THEN
	Stn710_DB.Alarm_count := 17;
END_IF

IF Stn710_DB.CC5_CLAMP.ErrHomeInterlock THEN
	Stn710_DB.Alarm_count := 18;
END_IF

IF Stn710_DB.CC5_CLAMP.ErrHomeTout THEN
	Stn710_DB.Alarm_count := 19;
END_IF

IF Stn710_DB.CC5_CLAMP.ErrWorkInterlock THEN
	Stn710_DB.Alarm_count := 20;
END_IF

IF Stn710_DB.CC5_CLAMP.ErrWorkTout THEN
	Stn710_DB.Alarm_count := 21;
END_IF

IF Stn710_DB.CC6_CLAMP.ErrHomeInterlock THEN
	Stn710_DB.Alarm_count := 22;
END_IF

IF Stn710_DB.CC6_CLAMP.ErrHomeTout THEN
	Stn710_DB.Alarm_count := 23;
END_IF

IF Stn710_DB.CC6_CLAMP.ErrWorkInterlock THEN
	Stn710_DB.Alarm_count := 24;
END_IF

IF Stn710_DB.CC6_CLAMP.ErrWorkTout THEN
	Stn710_DB.Alarm_count := 25;
END_IF

END_FUNCTION_BLOCK

// ---- GlobalTextList.TcGTLO
TEXTLIST GlobalTextList
  42 = 'Auto'
  8 = 'BUSY'
  357 = 'Button Palm'
  686 = 'CLAMP_1_HOME'
  638 = 'CLAMP_1_WORK'
  441 = 'CLAMP_2_HOME'
  102 = 'CLAMP_2_WORK'
  510 = 'CLAMP_3_HOME'
  453 = 'CLAMP_3_WORK'
  164 = 'CLAMP_4_HOME'
  720 = 'CLAMP_4_WORK'
  202 = 'CLAMP_5_HOME'
  862 = 'CLAMP_5_WORK'
  775 = 'CLAMP_6_HOME'
  610 = 'CLAMP_6_WORK'
  404 = 'CONTROL OFF'
  701 = 'CONTROL ON'
  226 = 'Cycle Start'
  363 = 'DOOR_DN'
  957 = 'DOOR_DOWN'
  151 = 'DOOR_UP'
  267 = 'DR DN'
  163 = 'DR DOWN'
  112 = 'DR UP'
  173 = 'Emergency Stop'
  503 = 'Fault Reset'
  942 = 'HOME'
  743 = 'Man'
  2 = 'MH_ROBOT'
  285 = 'Operator Palm'
  837 = 'Palm Button'
  366 = 'PART SENSORS'
  785 = 'POWER ON'
  599 = 'Power On'
  744 = 'START'
  570 = 'TR -20*'
  519 = 'TR 0*'
  681 = 'TR 45*'
  685 = 'TR 80*'
  966 = 'TR_-20'
  734 = 'TR_0'
  784 = 'TR_45'
  75 = 'TR_80'
  467 = 'TR_DOWN'
  338 = 'TR_UP'
  279 = 'TT 0*'
  639 = 'TT 180*'
  239 = 'TT_DOWN'
  295 = 'TT_FWD'
  871 = 'TT_REV'
  7 = 'WATER SPRAY'
  4 = 'WELD_ROBOT'
END_TEXTLIST

// ---- POUs/Library/Seq_list.TcTLO
TEXTLIST Seq_list
  0 = 'CYCLE START'
  10 = 'ROLLER DOOR_CLOSE'
  20 = 'TRUNION ROTATES -20*'
  30 = 'ROLLER DOOR OPEN'
  40 = 'OPERATOR LOAD 1st PART'
  50 = 'OPERATOR LOAD 2nd PART'
  60 = '1st, 3rd & 5th CLAMP CLOSE'
  70 = 'ROLLER DOOR_CLOSE'
  80 = 'TRUNION ROTATES 80*'
  90 = 'ROLLER DOOR OPEN'
  100 = 'OPERATOR LOAD_3rd_PART'
  110 = 'OPERATOR LOAD_4th_PART'
  120 = 'ROLLER DOOR_CLOSE'
  130 = '2nd, 4th & 6th CLAMP CLOSE'
  140 = 'TURNTABLE-180* AND TRUNION-0*'
  150 = 'Start WELD_Robot FOR WELD'
  160 = '1st, 3rd & 5th UNCLAMP'
  170 = 'ROLLER DOOR OPEN'
  180 = 'Start MH_Robot_1ST TIME'
  190 = 'TRUNION ROTATES 45*'
  200 = '2nd, 4th & 6th UNCLAMP '
  210 = 'Start MH_Robot_2ND TIME'
  220 = 'CYCLE COMPLETE'
  5 = 'WAIT FOR STATION HOME'
   = ''
END_TEXTLIST

// ---- POUs/Library/Alarm_list.TcTLO
TEXTLIST Alarm_list
  0 = 'No Alarm'
  1 = 'Emergency stop Pressed'
  2 = 'Home action Interlock error-CC1 \tClamp'
  3 = 'Home action timeout error-CC1 \tClamp'
  4 = 'Work action Interlock error-CC1 \tClamp'
  5 = 'Work action timeout error-CC1 \tClamp'
  6 = 'Home action Interlock error-CC2 \tClamp'
  7 = 'Home action timeout error-CC2\t Clamp'
  8 = 'Work action Interlock error-CC2 \tClamp'
  9 = 'Work action timeout error-CC2 \tClamp'
  10 = 'Home action Interlock error-CC3 \tClamp'
  11 = 'Home action timeout error-CC3\t Clamp'
  12 = 'Work action Interlock error-CC3 \tClamp'
  13 = 'Work action timeout error-CC3 \tClamp'
  14 = 'Home action Interlock error-CC4 \tClamp'
  15 = 'Home action timeout error-CC4\t Clamp'
  16 = 'Work action Interlock error-CC4 \tClamp'
  17 = 'Work action timeout error-CC4 \tClamp'
  18 = 'Home action Interlock error-CC5 \tClamp'
  19 = 'Home action timeout error-CC5\t Clamp'
  20 = 'Work action Interlock error-CC5 \tClamp'
  21 = 'Work action timeout error-CC5 \tClamp'
  22 = 'Home action Interlock error-CC6 \tClamp'
  23 = 'Home action timeout error-CC6\t Clamp'
  24 = 'Work action Interlock error-CC6 \tClamp'
  25 = 'Work action timeout error-CC6 \tClamp'
   = ''
END_TEXTLIST

// ---- VISUs/Visualization.TcVIS
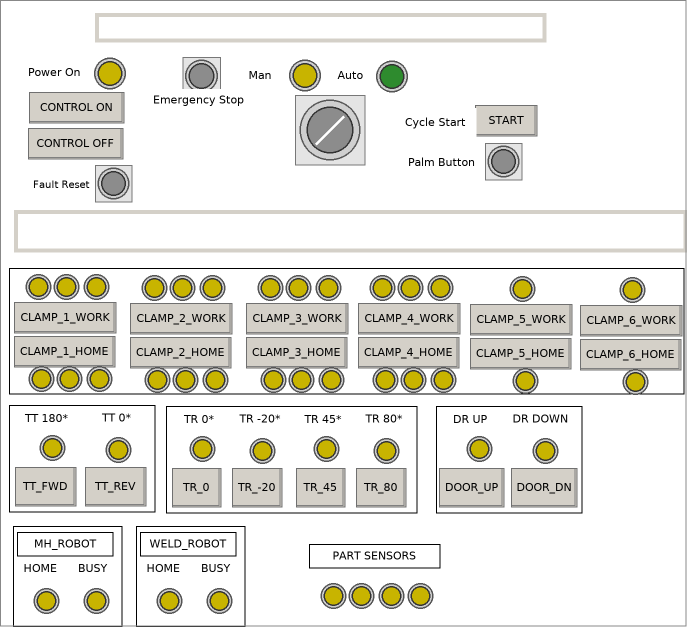
VISUALIZATION Visualization  // 687x627
    Rectangle (13,526 109x101)
    Rectangle (9,405 146x107)
    Rectangle (9,268 675x126)
    Lamp1 (85,55 50x37), variable: Outputs.qPower_On, style: Lamp-Lamp1-Yellow
    Button (29,92 95x31), "CONTROL ON", colour toggle: Inputs.iControl_On, input disabled if: Inputs.iEMR_Stop_PB
        toggle Inputs.iControl_On
    Textfield (24,58 61x29), "Power On"
    Button (28,128 95x31), "CONTROL OFF", colour toggle: Inputs.iControl_OFF
        toggle Inputs.iControl_Off
    RotarySwitch (295,95 70x70), variable: Inputs.iAuto_Manual, behaviour: TOGGLE, style: Switch-RotarySwitch-Gray
    Lamp1 (280,57 50x37), variable: Outputs.qStnMan, style: Lamp-Lamp1-Yellow
    Textfield (244,61 32x29), "Man"
    Lamp1 (367,58 50x37), variable: Outputs.qStnAuto, style: Lamp-Lamp1-Green
    Textfield (334,61 33x29), "Auto"
    Lamp1 (19,272 39x30), variable: Inputs.CC1_Clamp_1_Sensor_WP, style: Lamp-Lamp1-Yellow
    Button (14,302 102x31), "CLAMP_1_WORK", colour toggle: Stn710_DB.CC1_CLAMP.WorkCmd
        tap Stn710_DB.CC1_CLAMP.WorkCmd
    Button (14,336 101x31), "CLAMP_1_HOME", colour toggle: Stn710_DB.CC1_CLAMP.HomeCmd
        tap Stn710_DB.CC1_CLAMP.HomeCmd
    Lamp1 (47,272 39x30), variable: Inputs.CC1_Clamp_2_Sensor_WP, style: Lamp-Lamp1-Yellow
    Lamp1 (77,272 39x30), variable: Inputs.CC1_Clamp_3_Sensor_WP, style: Lamp-Lamp1-Yellow
    Lamp1 (22,364 39x30), variable: Inputs.CC1_Clamp_1_Sensor_HP, style: Lamp-Lamp1-Yellow
    Lamp1 (50,364 39x30), variable: Inputs.CC1_Clamp_2_Sensor_HP, style: Lamp-Lamp1-Yellow
    Lamp1 (80,364 39x30), variable: Inputs.CC1_Clamp_3_Sensor_HP, style: Lamp-Lamp1-Yellow
    PushSwitch (92,165 43x37), variable: Inputs.iResetFault, behaviour: TAP, style: Switch-PushSwitch-Gray
    Textfield (31,170 61x29), "Fault Reset"
    Lamp1 (135,273 39x30), variable: Inputs.CC2_Clamp_1_Sensor_WP, style: Lamp-Lamp1-Yellow
    Button (130,303 102x31), "CLAMP_2_WORK", colour toggle: Stn710_DB.CC2_CLAMP.WorkCmd
        tap Stn710_DB.CC2_CLAMP.WorkCmd
    Button (130,337 101x31), "CLAMP_2_HOME", colour toggle: Stn710_DB.CC2_CLAMP.HomeCmd
        tap Stn710_DB.CC2_CLAMP.HomeCmd
    Lamp1 (163,273 39x30), variable: Inputs.CC2_Clamp_2_Sensor_WP, style: Lamp-Lamp1-Yellow
    Lamp1 (193,273 39x30), variable: Inputs.CC2_Clamp_3_Sensor_WP, style: Lamp-Lamp1-Yellow
    Lamp1 (138,365 39x30), variable: Inputs.CC2_Clamp_1_Sensor_HP, style: Lamp-Lamp1-Yellow
    Lamp1 (166,365 39x30), variable: Inputs.CC2_Clamp_2_Sensor_HP, style: Lamp-Lamp1-Yellow
    Lamp1 (196,365 39x30), variable: Inputs.CC2_Clamp_3_Sensor_HP, style: Lamp-Lamp1-Yellow
    Lamp1 (251,273 39x30), variable: Inputs.CC3_Clamp_1_Sensor_WP, style: Lamp-Lamp1-Yellow
    Button (246,303 102x31), "CLAMP_3_WORK", colour toggle: Stn710_DB.CC3_CLAMP.WorkCmd
        tap Stn710_DB.CC3_CLAMP.WorkCmd
    Button (246,337 101x31), "CLAMP_3_HOME", colour toggle: Stn710_DB.CC3_CLAMP.HomeCmd
        tap Stn710_DB.CC3_CLAMP.HomeCmd
    Lamp1 (279,273 39x30), variable: Inputs.CC3_Clamp_2_Sensor_WP, style: Lamp-Lamp1-Yellow
    Lamp1 (309,273 39x30), variable: Inputs.CC3_Clamp_3_Sensor_WP, style: Lamp-Lamp1-Yellow
    Lamp1 (254,365 39x30), variable: Inputs.CC3_Clamp_1_Sensor_HP, style: Lamp-Lamp1-Yellow
    Lamp1 (282,365 39x30), variable: Inputs.CC3_Clamp_2_Sensor_HP, style: Lamp-Lamp1-Yellow
    Lamp1 (312,365 39x30), variable: Inputs.CC3_Clamp_3_Sensor_HP, style: Lamp-Lamp1-Yellow
    Lamp1 (363,273 39x30), variable: Inputs.CC4_Clamp_1_Sensor_WP, style: Lamp-Lamp1-Yellow
    Button (358,303 102x31), "CLAMP_4_WORK", colour toggle: Stn710_DB.CC4_CLAMP.WorkCmd
        tap Stn710_DB.CC4_CLAMP.WorkCmd
    Button (358,337 101x31), "CLAMP_4_HOME", colour toggle: Stn710_DB.CC4_CLAMP.HomeCmd
        tap Stn710_DB.CC4_CLAMP.HomeCmd
    Lamp1 (391,273 39x30), variable: Inputs.CC4_Clamp_2_Sensor_WP, style: Lamp-Lamp1-Yellow
    Lamp1 (421,273 39x30), variable: Inputs.CC4_Clamp_3_Sensor_WP, style: Lamp-Lamp1-Yellow
    Lamp1 (366,365 39x30), variable: Inputs.CC4_Clamp_1_Sensor_HP, style: Lamp-Lamp1-Yellow
    Lamp1 (394,365 39x30), variable: Inputs.CC4_Clamp_2_Sensor_HP, style: Lamp-Lamp1-Yellow
    Lamp1 (424,365 39x30), variable: Inputs.CC4_Clamp_3_Sensor_HP, style: Lamp-Lamp1-Yellow
    Button (470,304 102x31), "CLAMP_5_WORK", colour toggle: Stn710_DB.CC5_CLAMP.WorkCmd
        tap Stn710_DB.CC5_CLAMP.WorkCmd
    Button (470,338 101x31), "CLAMP_5_HOME", colour toggle: Stn710_DB.CC5_CLAMP.HomeCmd
        tap Stn710_DB.CC5_CLAMP.HomeCmd
    Lamp1 (503,274 39x30), variable: Inputs.CC5_Clamp_1_Sensor_WP, style: Lamp-Lamp1-Yellow
    Lamp1 (506,366 39x30), variable: Inputs.CC5_Clamp_1_Sensor_HP, style: Lamp-Lamp1-Yellow
    Lamp1 (613,275 39x30), variable: Inputs.CC6_Clamp_1_Sensor_WP, style: Lamp-Lamp1-Yellow
    Button (580,305 102x31), "CLAMP_6_WORK", colour toggle: Stn710_DB.CC6_CLAMP.WorkCmd
        tap Stn710_DB.CC6_CLAMP.WorkCmd
    Button (580,339 101x31), "CLAMP_6_HOME", colour toggle: Stn710_DB.CC6_CLAMP.HomeCmd
        tap Stn710_DB.CC6_CLAMP.HomeCmd
    Lamp1 (616,367 39x30), variable: Inputs.CC6_Clamp_1_Sensor_HP, style: Lamp-Lamp1-Yellow
    Button (15,467 61x39), "TT_FWD", colour toggle: Stn710_DB.M_TT_CW
        tap Stn710_DB.M_TT_CW
    Button (85,467 61x39), "TT_REV", colour toggle: Stn710_DB.M_TT_CCW
        tap Stn710_DB.M_TT_CCW
    Lamp1 (33,433 39x30), variable: Stn710_DB.M_TT_FwdSens, style: Lamp-Lamp1-Yellow
    Lamp1 (99,435 39x30), variable: Stn710_DB.M_TT_RevSens, style: Lamp-Lamp1-Yellow
    Textfield (16,409 61x19), "TT 180*"
    Textfield (86,408 61x20), "TT 0*"
    Rectangle (166,406 251x107)
    Button (172,468 49x39), "TR_0", colour toggle: Stn710_DB.M_TR_0_CMD
        tap Stn710_DB.M_TR_0_CMD
    Button (232,468 50x39), "TR_-20", colour toggle: Stn710_DB.M_TR_20_CMD
        tap Stn710_DB.M_TR_20_CMD
    Lamp1 (183,434 39x30), variable: Stn710_DB.M_TR_0_FB, style: Lamp-Lamp1-Yellow
    Lamp1 (243,436 39x30), variable: Stn710_DB.M_TR_20_FB, style: Lamp-Lamp1-Yellow
    Textfield (171,410 56x19), "TR 0*"
    Textfield (235,409 50x20), "TR -20*"
    PushSwitchLed (176,57 51x38), variable: Inputs.iEMR_Stop_PB, behaviour: TOGGLE, style: Switch-PushSwitchLed-Gray
    Textfield (145,89 107x22), "Emergency Stop"
    Rectangle (436,406 146x107)
    Button (439,468 65x39), "DOOR_UP", colour toggle: Stn710_DB.M_DR_UP
        tap Stn710_DB.M_DR_UP
    Button (511,468 66x39), "DOOR_DN", colour toggle: Stn710_DB.M_DR_DOWN
        tap Stn710_DB.M_DR_DOWN
    Lamp1 (460,434 39x30), variable: Stn710_DB.M_DR_UPSens, style: Lamp-Lamp1-Yellow
    Lamp1 (526,436 39x30), variable: Stn710_DB.M_DR_DNSens, style: Lamp-Lamp1-Yellow
    Textfield (443,410 54x19), "DR UP"
    Textfield (507,409 67x20), "DR DOWN"
    Rectangle (17,532 96x24), "MH_ROBOT"
    Textfield (19,559 43x19), "HOME"
    Textfield (73,559 39x19), "BUSY"
    Lamp1 (27,586 39x30), variable: Stn710_DB.MH_RobotHome, style: Lamp-Lamp1-Yellow
    Lamp1 (77,586 39x30), variable: Stn710_DB.MH_RobotBusy, style: Lamp-Lamp1-Yellow
    Rectangle (136,526 109x101)
    Rectangle (140,532 96x24), "WELD_ROBOT"
    Textfield (142,559 43x19), "HOME"
    Textfield (196,559 39x19), "BUSY"
    Lamp1 (150,586 39x30), variable: Stn710_DB.WELD_RobotHome, style: Lamp-Lamp1-Yellow
    Lamp1 (200,586 39x30), variable: Stn710_DB.WELD_RobotBusy, style: Lamp-Lamp1-Yellow
    Textfield (14,210 673x42), text list: 'Seq_list', text index: Auto_Seq_DB.MStep
    Lamp1 (314,581 39x30), variable: Auto_Seq_DB.Part_Sensor1, style: Lamp-Lamp1-Yellow
    Lamp1 (342,581 39x30), variable: Auto_Seq_DB.Part_Sensor2, style: Lamp-Lamp1-Yellow
    Lamp1 (372,581 39x30), variable: Auto_Seq_DB.Part_Sensor3, style: Lamp-Lamp1-Yellow
    Rectangle (309,544 131x24), "PART SENSORS"
    Lamp1 (401,581 39x30), variable: Auto_Seq_DB.Part_Sensor4, style: Lamp-Lamp1-Yellow
    Button (475,105 62x31), "START", colour toggle: Inputs.iCycle_start
        tap Inputs.iCycle_start
    Textfield (401,148 81x29), "Palm Button"
    PushSwitch (482,143 43x37), variable: Inputs.iPalm_Button, behaviour: TAP, style: Switch-PushSwitch-Gray
    Textfield (395,108 81x29), "Cycle Start"
    Textfield (295,410 56x19), "TR 45*"
    Button (296,468 49x39), "TR_45", colour toggle: Stn710_DB.M_TR_45_CMD
        tap Stn710_DB.M_TR_45_CMD
    Button (356,468 50x39), "TR_80", colour toggle: Stn710_DB.M_TR_80_CMD
        tap Stn710_DB.M_TR_80_CMD
    Lamp1 (307,434 39x30), variable: Stn710_DB.M_TR_45_FB, style: Lamp-Lamp1-Yellow
    Lamp1 (367,436 39x30), variable: Stn710_DB.M_TR_80_FB, style: Lamp-Lamp1-Yellow
    Textfield (359,409 50x20), "TR 80*"
    Textfield (95,13 451x29), text list: 'Alarm_list', text index: Stn710_DB.Alarm_count
END_VISUALIZATION
